// TIA Portal project "DATN" (V17)

(* hardware
DEVICE "S7-1200 station_1"  S7-1200 Station
   slot 0: "Rack_0"  S7-1200 Rack  Rack  V1.0
   slot 1: "PLC_1"  CPU 1214C DC/DC/DC  6ES7 214-1AG40-0XB0  V4.5
DEVICE "HMI_1"  KTP700 Basic PN
   slot 0: "HMI_1"  KTP700 Basic PN  6AV2 123-2GB03-0AX0  17.0.0.0
   slot 1: "HMI_RT_1"  KTP700 Basic PN  6AV2 123-2GB03-0AX0  17.0.0.0
   slot 5: "HMI_1.IE_CP_1"  PROFINET Interface  17.0.0.0
      slot 1: "PROFINET Interface_1"  PROFINET Interface
         slot 1: "Port_1"  Port
*)

// ===== PLC "PLC_1"  CPU 1214C DC/DC/DC =====

VAR_GLOBAL   // PLC tag table "Default tag table"
   "Tag_1" AT %M53.0 : Bool;
   "Reset_ctu_alarm" AT %M53.3 : Bool;
   "Tag_2" AT %M53.1 : Bool;
   "Tag_3" AT %M53.2 : Bool;
   "Error_lamp_alarm" AT %M53.4 : Bool;
   "time_up_maintenance" AT %M53.5 : Bool;
   "Alarm_not_product" AT %M53.6 : Bool;
   "Tag_4" AT %M100.0 : Bool;
   "Tag_5" AT %M100.1 : Bool;
   "Tag_6" AT %Q0.0 : Bool;
   "over_memory" AT %M54.0 : Bool;
   "stop_Sys_alarm" AT %M54.1 : Bool;
END_VAR

VAR_GLOBAL   // PLC tag table "Sensor"
   "Sensor_1" AT %I0.3 : Bool;
   "Sensor_2" AT %I0.4 : Bool;
   "Sensor_3" AT %I0.5 : Bool;
   "Sensor_4" AT %I0.6 : Bool;
   "Sensor_5" AT %I0.7 : Bool;
   "Sensor_Detech" AT %I0.2 : Bool;
END_VAR

VAR_GLOBAL   // PLC tag table "Output"
   "cylinder_1" AT %Q0.1 : Bool;
   "cylinder_2" AT %Q1.1 : Bool;
   "cylinder_3" AT %Q0.3 : Bool;
   "cylinder_4" AT %Q0.4 : Bool;
   "cylinder_5" AT %Q0.5 : Bool;
   "converyor" AT %Q1.0 : Bool;
   "led_error" AT %Q0.6 : Bool;
END_VAR

VAR_GLOBAL   // PLC tag table "Input_control"
   "Start" AT %I0.0 : Bool;
   "Stop" AT %I0.1 : Bool;
END_VAR

VAR_GLOBAL   // PLC tag table "State_system"
   "State_all" AT %M10.0 : Bool;
   "State_auto" AT %M10.1 : Bool;
END_VAR

VAR_GLOBAL   // PLC tag table "HMI"
   "hmi_manu_cylinder_1" AT %M10.3 : Bool;
   "hmi_manu_cylinder_2" AT %M10.4 : Bool;
   "hmi_manu_cylinder_3" AT %M10.5 : Bool;
   "hmi_manu_cylinder_4" AT %M10.6 : Bool;
   "hmi_manu_cylinder_5" AT %M10.7 : Bool;
   "hmi_active_count" AT %M11.0 : Bool;
   "HMI_ALARM" AT %M11.1 : Bool;
   "hmi_manu_conveyor" AT %M10.2 : Bool;
   "HMI_START" AT %M11.2 : Bool;
   "HMI_STOP" AT %M11.3 : Bool;
   "hmi_reset_count" AT %M11.4 : Bool;
   "hmi_problem_handled" AT %M11.5 : Bool;
   "hmi_reset_data" AT %M11.6 : Bool;
END_VAR

VAR_GLOBAL   // PLC tag table "Alarm"
   "Alarm1" AT %MW20 : Word;
   "Alarm1_Bit8_Motor_Fault" AT %M20.0 : Bool;   // Alarm motor Fault
   "Alarm1_Bit9_cylinder1_Fault" AT %M20.1 : Bool;   // Alarm cylinder1 Fault
   "Alarm1_Bit10_cylinder2_Fault" AT %M20.2 : Bool;   // Alarm cylinder2 Fault
   "Alarm1_Bit11_cylinder3_Fault" AT %M20.3 : Bool;   // Alarm cylinder3 Fault
   "Alarm1_Bit12_cylinder4_Fault" AT %M20.4 : Bool;   // Alarm cylinder4 Fault
   "Alarm1_Bit13_cylinder5_Fault" AT %M20.5 : Bool;   // Alarm cylinder5 Fault
   "Alarm1_Bit14" AT %M20.6 : Bool;   // Spare
   "Alarm1_Bit15" AT %M20.7 : Bool;   // Spare
   "Alarm1_Bit0" AT %M21.0 : Bool;   // Spare
   "Alarm1_Bit1" AT %M21.1 : Bool;   // Spare
   "Alarm1_Bit2" AT %M21.2 : Bool;   // Spare
   "Alarm1_Bit3" AT %M21.3 : Bool;   // Spare
   "Alarm_over_memory" AT %M21.4 : Bool;   // over memory
   "Alarm_emergence_stop_web" AT %M21.5 : Bool;   // emergence stop
   "Alarm_camera_error" AT %M21.6 : Bool;   // camera error
   "Alarm_maintenance_time" AT %M21.7 : Bool;   // up to maintenance time
END_VAR

VAR_GLOBAL   // PLC tag table "Simulater"
   "Sim_motor_tripped" AT %M52.0 : Bool;
   "Sim_cylinder1_tripped" AT %M52.1 : Bool;
   "Sim_cylinder2_tripped" AT %M52.2 : Bool;
   "Sim_cylinder3_tripped" AT %M52.3 : Bool;
   "Sim_cylinder4_tripped" AT %M52.4 : Bool;
   "Sim_cylinder5_tripped" AT %M52.5 : Bool;
END_VAR

DATA_BLOCK "Array_threading"   // DB1
{ S7_Optimized_Access := 'FALSE' }
VERSION : 0.1
   VAR
      array_threading_1 : Array[0..20] of Int;
      array_threading_2 : Array[0..20] of Int;
      array_threading_3 : Array[0..20] of Int;
      array_threading_4 : Array[0..20] of Int;
      array_threading_5 : Array[0..20] of Int;
      last_run_1 : Bool;
      last_run_2 : Bool;
      last_run_3 : Bool;
      last_run_4 : Bool;
      last_run_5 : Bool;
   END_VAR
BEGIN
END_DATA_BLOCK

DATA_BLOCK "Data_webcam"   // DB7
{ S7_Optimized_Access := 'FALSE' }
VERSION : 0.1
   VAR
      new_position : Int;
      save_new_position : Bool;
      state_camera : Bool := true;
      alarm_error : Bool;
      state_auto : Bool;
      last_state_sensor_1 : Bool;
      last_state_sensor_2 : Bool;
      last_state_sensor_3 : Bool;
      last_state_sensor_4 : Bool;
      last_state_sensor_5 : Bool;
      last_save_new_position : Bool;
   END_VAR
BEGIN
END_DATA_BLOCK

DATA_BLOCK "Data_count_Position"   // DB8
{ S7_Optimized_Access := 'FALSE' }
VERSION : 0.1
   VAR
      Adress_1 : Real;
      Adress_2 : Real;
      Adress_3 : Real;
      Adress_4 : Real;
      Adress_5 : Real;
      Adress_6 : Real;
   END_VAR
BEGIN
END_DATA_BLOCK

DATA_BLOCK "Data_alarm"   // DB17
{ S7_Optimized_Access := 'FALSE' }
VERSION : 0.1
   VAR
      Motor_tripped : Bool;
      Cylinder1_tripped : Bool;
      Cylinder2_tripped : Bool;
      Cylinder3_tripped : Bool;
      Cylinder4_tripped : Bool;
      Cylinder5_tripped : Bool;
      Camera_tripped : Bool;
      Time_to_Maintenance : DInt;
   END_VAR
BEGIN
END_DATA_BLOCK

DATA_BLOCK "state_to_webserver"   // DB22
{ S7_Optimized_Access := 'FALSE' }
VERSION : 0.1
   VAR
      state_sensor_1 : Bool;
      state_sensor_2 : Bool;
      state_sensor_3 : Bool;
      state_sensor_4 : Bool;
      state_sensor_5 : Bool;
      state_sensor_detech : Bool;
      state_emergency_stop : Bool;
      state_cylinder_1 : Int;
      state_cylinder_2 : Int;
      state_cylinder_3 : Int;
      state_cylinder_4 : Int;
      state_cylinder_5 : Int;
      state_motor : Int;
      state_auto : Int;
   END_VAR
BEGIN
END_DATA_BLOCK

// folder: System blocks/Program resources

DATA_BLOCK "IEC_Timer_0_DB"   // DB2
{ S7_Optimized_Access := 'TRUE' }
AUTHOR : Simatic
FAMILY : IEC
NAME : IEC_TMR
VERSION : 1.0
// stored: InstanceOfName IEC_TIMER
"IEC_TIMER"
BEGIN
END_DATA_BLOCK

DATA_BLOCK "IEC_Timer_0_DB_1"   // DB3
{ S7_Optimized_Access := 'TRUE' }
AUTHOR : Simatic
FAMILY : IEC
NAME : IEC_TMR
VERSION : 1.0
// stored: InstanceOfName IEC_TIMER
"IEC_TIMER"
BEGIN
END_DATA_BLOCK

DATA_BLOCK "IEC_Timer_0_DB_2"   // DB4
{ S7_Optimized_Access := 'TRUE' }
AUTHOR : Simatic
FAMILY : IEC
NAME : IEC_TMR
VERSION : 1.0
// stored: InstanceOfName IEC_TIMER
"IEC_TIMER"
BEGIN
END_DATA_BLOCK

DATA_BLOCK "IEC_Timer_0_DB_3"   // DB5
{ S7_Optimized_Access := 'TRUE' }
AUTHOR : Simatic
FAMILY : IEC
NAME : IEC_TMR
VERSION : 1.0
// stored: InstanceOfName IEC_TIMER
"IEC_TIMER"
BEGIN
END_DATA_BLOCK

DATA_BLOCK "IEC_Timer_0_DB_4"   // DB6
{ S7_Optimized_Access := 'TRUE' }
AUTHOR : Simatic
FAMILY : IEC
NAME : IEC_TMR
VERSION : 1.0
// stored: InstanceOfName IEC_TIMER
"IEC_TIMER"
BEGIN
END_DATA_BLOCK

DATA_BLOCK "IEC_Counter_0_DB"   // DB9
{ S7_Optimized_Access := 'FALSE' }
AUTHOR : Simatic
FAMILY : IEC
NAME : CNTR
VERSION : 1.0
// stored: InstanceOfName IEC_COUNTER
"IEC_COUNTER"
BEGIN
END_DATA_BLOCK

DATA_BLOCK "IEC_Counter_0_DB_1"   // DB10
{ S7_Optimized_Access := 'TRUE' }
AUTHOR : Simatic
FAMILY : IEC
NAME : CNTR
VERSION : 1.0
// stored: InstanceOfName IEC_COUNTER
"IEC_COUNTER"
BEGIN
END_DATA_BLOCK

DATA_BLOCK "IEC_Counter_0_DB_2"   // DB11
{ S7_Optimized_Access := 'TRUE' }
AUTHOR : Simatic
FAMILY : IEC
NAME : CNTR
VERSION : 1.0
// stored: InstanceOfName IEC_COUNTER
"IEC_COUNTER"
BEGIN
END_DATA_BLOCK

DATA_BLOCK "IEC_Counter_0_DB_3"   // DB12
{ S7_Optimized_Access := 'TRUE' }
AUTHOR : Simatic
FAMILY : IEC
NAME : CNTR
VERSION : 1.0
// stored: InstanceOfName IEC_COUNTER
"IEC_COUNTER"
BEGIN
END_DATA_BLOCK

DATA_BLOCK "IEC_Counter_0_DB_4"   // DB13
{ S7_Optimized_Access := 'TRUE' }
AUTHOR : Simatic
FAMILY : IEC
NAME : CNTR
VERSION : 1.0
// stored: InstanceOfName IEC_COUNTER
"IEC_COUNTER"
BEGIN
END_DATA_BLOCK

DATA_BLOCK "IEC_Timer_0_DB_7"   // DB14
{ S7_Optimized_Access := 'TRUE' }
AUTHOR : Simatic
FAMILY : IEC
NAME : IEC_TMR
VERSION : 1.0
// stored: InstanceOfName IEC_TIMER
"IEC_TIMER"
BEGIN
END_DATA_BLOCK

DATA_BLOCK "IEC_Counter_0_DB_6"   // DB20
{ S7_Optimized_Access := 'TRUE' }
AUTHOR : SIMATIC
FAMILY : IEC
NAME : DCNTR
VERSION : 1.2
// stored: InstanceOfName IEC_DCOUNTER
"IEC_DCOUNTER"
BEGIN
END_DATA_BLOCK

DATA_BLOCK "IEC_Timer_0_DB_9"   // DB21
{ S7_Optimized_Access := 'TRUE' }
AUTHOR : Simatic
FAMILY : IEC
NAME : IEC_TMR
VERSION : 1.0
// stored: InstanceOfName IEC_TIMER
"IEC_TIMER"
BEGIN
END_DATA_BLOCK

// folder: (top level)

FUNCTION "Auto" : Void   // FC1, LAD
{ S7_Optimized_Access := 'TRUE' }
VERSION : 0.1
   VAR_INPUT
      error_alarm : Bool;
      new_position : Int;
      save_new_position : Bool;
      reset_data : Bool;
      sensor_1 : Bool;
      sensor_2 : Bool;
      sensor_3 : Bool;
      sensor_4 : Bool;
      sensor_5 : Bool;
   END_VAR
   VAR_OUTPUT
      cylinder_1 : Bool;
      cylinder_2 : Bool;
      cylinder_3 : Bool;
      cylinder_4 : Bool;
      cylinder_5 : Bool;
      over_memory : Bool;
   END_VAR
   VAR_TEMP
      loop_element : Int;
      last_child_array_1 : Int;
      last_child_array_2 : Int;
      last_child_array_3 : Int;
      last_child_array_4 : Int;
      last_child_array_5 : Int;
      trigger_sensor_1 : Bool;
      trigger_sensor_2 : Bool;
      trigger_sensor_3 : Bool;
      trigger_sensor_4 : Bool;
      trigger_sensor_5 : Bool;
   END_VAR
BEGIN

REGION Network 1 (SCL): Program main
   // chuong trinh dieu khien
   // ========================
   // Reset trạng thái khi save_new_position = 0 hoặc cảm biến = 0
   // ========================
   IF #save_new_position = FALSE THEN
       "Data_webcam".last_save_new_position := FALSE;
   END_IF;

   IF #sensor_1 = FALSE THEN
       "Data_webcam".last_state_sensor_1 := FALSE;
   END_IF;

   IF #sensor_2 = FALSE THEN
       "Data_webcam".last_state_sensor_2 := FALSE;
   END_IF;

   IF #sensor_3 = FALSE THEN
       "Data_webcam".last_state_sensor_3 := FALSE;
   END_IF;

   IF #sensor_4 = FALSE THEN
       "Data_webcam".last_state_sensor_4 := FALSE;
   END_IF;

   IF #sensor_5 = FALSE THEN
       "Data_webcam".last_state_sensor_5 := FALSE;
   END_IF;

   // ========================
   // Xử lý khi có sản phẩm mới
   // ========================
   IF (#save_new_position = TRUE) AND ("Data_webcam".last_save_new_position = FALSE) AND (#error_alarm = False) THEN
       "Data_webcam".last_save_new_position := TRUE;

       // Tìm vị trí cuối cùng của mỗi mảng
       #last_child_array_1 := -1;
       #last_child_array_2 := -1;
       #last_child_array_3 := -1;
       #last_child_array_4 := -1;
       #last_child_array_5 := -1;

       FOR #loop_element := 0 TO 20 DO
           IF ("Array_threading".array_threading_1[#loop_element] = 1) OR ("Array_threading".array_threading_1[#loop_element] = 2) THEN
               #last_child_array_1 := #loop_element;
           END_IF;
           IF ("Array_threading".array_threading_2[#loop_element] = 1) OR ("Array_threading".array_threading_2[#loop_element] = 2) THEN
               #last_child_array_2 := #loop_element;
           END_IF;
           IF ("Array_threading".array_threading_3[#loop_element] = 1) OR ("Array_threading".array_threading_3[#loop_element] = 2) THEN
               #last_child_array_3 := #loop_element;
           END_IF;
           IF ("Array_threading".array_threading_4[#loop_element] = 1) OR ("Array_threading".array_threading_4[#loop_element] = 2) THEN
               #last_child_array_4 := #loop_element;
           END_IF;
           IF ("Array_threading".array_threading_5[#loop_element] = 1) OR ("Array_threading".array_threading_5[#loop_element] = 2) THEN
               #last_child_array_5 := #loop_element;
           END_IF;
       END_FOR;

       // Gán vị trí mới (tránh tràn mảng)
       CASE #new_position OF
           1:
               IF #last_child_array_1 < 20 THEN
                   "Array_threading".array_threading_1[#last_child_array_1 + 1] := 1;
               END_IF;

           2:
               IF #last_child_array_1 < 20 AND #last_child_array_2 < 20 THEN
                   "Array_threading".array_threading_1[#last_child_array_1 + 1] := 2;
                   "Array_threading".array_threading_2[#last_child_array_2 + 1] := 1;
               END_IF;

           3:
               IF #last_child_array_1 < 20 AND #last_child_array_2 < 20 AND #last_child_array_3 < 20 THEN
                   "Array_threading".array_threading_1[#last_child_array_1 + 1] := 2;
                   "Array_threading".array_threading_2[#last_child_array_2 + 1] := 2;
                   "Array_threading".array_threading_3[#last_child_array_3 + 1] := 1;
               END_IF;

           4:
               IF #last_child_array_1 < 20 AND #last_child_array_2 < 20 AND
                   #last_child_array_3 < 20 AND #last_child_array_4 < 20 THEN
                   "Array_threading".array_threading_1[#last_child_array_1 + 1] := 2;
                   "Array_threading".array_threading_2[#last_child_array_2 + 1] := 2;
                   "Array_threading".array_threading_3[#last_child_array_3 + 1] := 2;
                   "Array_threading".array_threading_4[#last_child_array_4 + 1] := 1;
               END_IF;

           5:
               IF #last_child_array_1 < 20 AND #last_child_array_2 < 20 AND
                   #last_child_array_3 < 20 AND #last_child_array_4 < 20 AND
                   #last_child_array_5 < 20 THEN
                   "Array_threading".array_threading_1[#last_child_array_1 + 1] := 2;
                   "Array_threading".array_threading_2[#last_child_array_2 + 1] := 2;
                   "Array_threading".array_threading_3[#last_child_array_3 + 1] := 2;
                   "Array_threading".array_threading_4[#last_child_array_4 + 1] := 2;
                   "Array_threading".array_threading_5[#last_child_array_5 + 1] := 1;
               END_IF;

           6:
               IF #last_child_array_1 < 20 AND #last_child_array_2 < 20 AND
                   #last_child_array_3 < 20 AND #last_child_array_4 < 20 AND
                   #last_child_array_5 < 20 THEN
                   "Array_threading".array_threading_1[#last_child_array_1 + 1] := 2;
                   "Array_threading".array_threading_2[#last_child_array_2 + 1] := 2;
                   "Array_threading".array_threading_3[#last_child_array_3 + 1] := 2;
                   "Array_threading".array_threading_4[#last_child_array_4 + 1] := 2;
                   "Array_threading".array_threading_5[#last_child_array_5 + 1] := 2;
               END_IF;
       END_CASE;
   END_IF;

   // Báo tràn bộ nhớ phân loại
   IF #last_child_array_1 = 20 OR #last_child_array_2 = 20 OR
       #last_child_array_3 = 20 OR #last_child_array_4 = 20 OR
       #last_child_array_5 = 20 THEN
       #over_memory := TRUE;
   END_IF;

   // ========================
   // Xử lý từng cảm biến khi phát hiện sản phẩm
   // ========================
   // ==== SENSOR 1 ====
   IF (#sensor_1 = TRUE) AND (#sensor_1 <> "Data_webcam".last_state_sensor_1) AND "Array_threading".last_run_1 = FALSE THEN
       // Set trigger cho TOF

       IF "Array_threading".array_threading_1[0] = 1 THEN
           #trigger_sensor_1 := TRUE;
       END_IF;

       FOR #loop_element := 0 TO 19 DO
           "Array_threading".array_threading_1[#loop_element] := "Array_threading".array_threading_1[#loop_element + 1];
       END_FOR;
       "Array_threading".array_threading_1[20] := 0;
       "Data_webcam".last_state_sensor_1 := TRUE;
   END_IF;

   // ==== SENSOR 2 ====
   IF (#sensor_2 = TRUE) AND (#sensor_2 <> "Data_webcam".last_state_sensor_2) AND "Array_threading".last_run_2 = FALSE THEN
       IF "Array_threading".array_threading_2[0] = 1 THEN
           #trigger_sensor_2 := TRUE;
       END_IF;

       FOR #loop_element := 0 TO 19 DO
           "Array_threading".array_threading_2[#loop_element] := "Array_threading".array_threading_2[#loop_element + 1];
       END_FOR;
       "Array_threading".array_threading_2[20] := 0;
       "Data_webcam".last_state_sensor_2 := TRUE;
   END_IF;

   // ==== SENSOR 3 ====
   IF (#sensor_3 = TRUE) AND (#sensor_3 <> "Data_webcam".last_state_sensor_3) AND "Array_threading".last_run_3 = FALSE THEN
       IF "Array_threading".array_threading_3[0] = 1 THEN
           #trigger_sensor_3 := TRUE;
       END_IF;

       FOR #loop_element := 0 TO 19 DO
           "Array_threading".array_threading_3[#loop_element] := "Array_threading".array_threading_3[#loop_element + 1];
       END_FOR;
       "Array_threading".array_threading_3[20] := 0;
       "Data_webcam".last_state_sensor_3 := TRUE;
   END_IF;

   // ==== SENSOR 4 ====
   IF (#sensor_4 = TRUE) AND (#sensor_4 <> "Data_webcam".last_state_sensor_4) AND "Array_threading".last_run_4 = FALSE THEN
       IF "Array_threading".array_threading_4[0] = 1 THEN
           #trigger_sensor_4 := TRUE;
       END_IF;

       FOR #loop_element := 0 TO 19 DO
           "Array_threading".array_threading_4[#loop_element] := "Array_threading".array_threading_4[#loop_element + 1];
       END_FOR;
       "Array_threading".array_threading_4[20] := 0;
       "Data_webcam".last_state_sensor_4 := TRUE;
   END_IF;

   // ==== SENSOR 5 ====
   IF (#sensor_5 = TRUE) AND (#sensor_5 <> "Data_webcam".last_state_sensor_5) AND "Array_threading".last_run_5 = FALSE THEN
       IF "Array_threading".array_threading_5[0] = 1 THEN
           #trigger_sensor_5 := TRUE;
       END_IF;

       FOR #loop_element := 0 TO 19 DO
           "Array_threading".array_threading_5[#loop_element] := "Array_threading".array_threading_5[#loop_element + 1];
       END_FOR;
       "Array_threading".array_threading_5[20] := 0;
       "Data_webcam".last_state_sensor_5 := TRUE;
   END_IF;

   // ======== TIMER ON DELAY ========
   "IEC_Timer_0_DB".TOF(IN:=#trigger_sensor_1,PT:=T#3s);
   "IEC_Timer_0_DB_1".TOF(IN:=#trigger_sensor_2,PT:=T#3s);
   "IEC_Timer_0_DB_2".TOF(IN :=#trigger_sensor_3,PT := T#3s);
   "IEC_Timer_0_DB_3".TOF(IN :=#trigger_sensor_4,PT:=T#3s);
   "IEC_Timer_0_DB_4".TOF(IN:=#trigger_sensor_5,PT:=T#3s);

   IF ("IEC_Timer_0_DB".ET >= T#1s) AND ("IEC_Timer_0_DB".ET < T#2s) THEN
       #cylinder_1 := TRUE;
   ELSE
       #cylinder_1 := FALSE;
   END_IF;

   IF ("IEC_Timer_0_DB_1".ET >= T#1s) AND ("IEC_Timer_0_DB_1".ET < T#2s) THEN
       #cylinder_2 := TRUE;
   ELSE
       #cylinder_2 := FALSE;
   END_IF;

   IF ("IEC_Timer_0_DB_2".ET >= T#1s) AND ("IEC_Timer_0_DB_2".ET < T#2s) THEN
       #cylinder_3 := TRUE;
   ELSE
       #cylinder_3 := FALSE;
   END_IF;

   IF ("IEC_Timer_0_DB_3".ET >= T#1s) AND ("IEC_Timer_0_DB_3".ET < T#2s) THEN
       #cylinder_4 := TRUE;
   ELSE
       #cylinder_4 := FALSE;
   END_IF;

   IF ("IEC_Timer_0_DB_4".ET >= T#1s) AND ("IEC_Timer_0_DB_4".ET < T#2s) THEN
       #cylinder_5 := TRUE;
   ELSE
       #cylinder_5 := FALSE;
   END_IF;


   // ======== RESET DATA  ========
   IF #reset_data = TRUE THEN
       FOR #loop_element := 0 TO 20 DO
           "Array_threading".array_threading_1[#loop_element] := 0;
           "Array_threading".array_threading_2[#loop_element] := 0;
           "Array_threading".array_threading_3[#loop_element] := 0;
           "Array_threading".array_threading_4[#loop_element] := 0;
           "Array_threading".array_threading_5[#loop_element] := 0;
       END_FOR;
   END_IF;
END_REGION
END_FUNCTION

FUNCTION "Manual" : Void   // FC2, LAD
{ S7_Optimized_Access := 'TRUE' }
VERSION : 0.1
   VAR_INPUT
      control_conveyor : Bool;
      control_cylinder_1 : Bool;
      control_cylinder_2 : Bool;
      control_cylinder_3 : Bool;
      control_cylinder_4 : Bool;
      control_cylinder_5 : Bool;
   END_VAR
   VAR_OUTPUT
      conveyor : Bool;
      cylinder_1 : Bool;
      cylinder_2 : Bool;
      cylinder_3 : Bool;
      cylinder_4 : Bool;
      cylinder_5 : Bool;
   END_VAR
BEGIN

REGION Network 1: Program manual conveyor
   // chuong trinh dieu khien bang tay bang tai
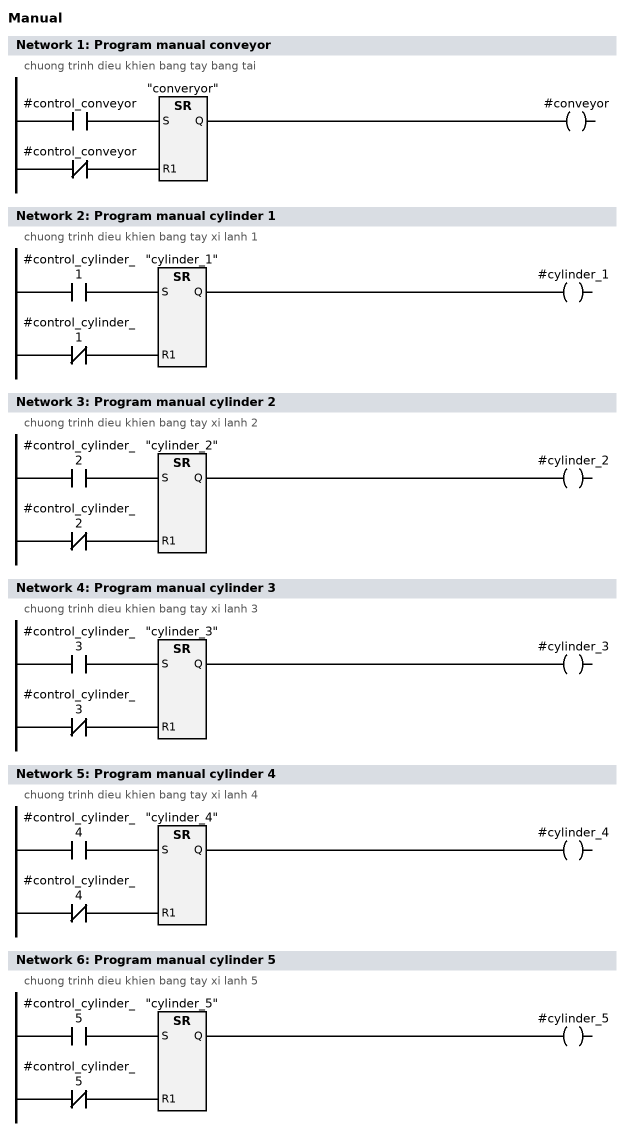
   RUNG wire#powerrail
      Contact( #control_conveyor )
      S_SR(operand := "converyor", r1 := wire#w1)
      Coil( #conveyor )
   END_RUNG
   RUNG wire#powerrail
      I_Contact( #control_conveyor )
   END_RUNG wire#w1
   // the same network as SCL:
   IF #control_conveyor THEN
       "converyor" := TRUE;   // SR flip-flop
   END_IF;
   IF NOT #control_conveyor THEN "converyor" := FALSE; END_IF;
   #conveyor := "converyor";
END_REGION

REGION Network 2: Program manual cylinder 1
   // chuong trinh dieu khien bang tay xi lanh 1
   RUNG wire#powerrail
      Contact( #control_cylinder_1 )
      S_SR(operand := "cylinder_1", r1 := wire#w1)
      Coil( #cylinder_1 )
   END_RUNG
   RUNG wire#powerrail
      I_Contact( #control_cylinder_1 )
   END_RUNG wire#w1
   // the same network as SCL:
   IF #control_cylinder_1 THEN
       "cylinder_1" := TRUE;   // SR flip-flop
   END_IF;
   IF NOT #control_cylinder_1 THEN "cylinder_1" := FALSE; END_IF;
   #cylinder_1 := "cylinder_1";
END_REGION

REGION Network 3: Program manual cylinder 2
   // chuong trinh dieu khien bang tay xi lanh 2
   RUNG wire#powerrail
      Contact( #control_cylinder_2 )
      S_SR(operand := "cylinder_2", r1 := wire#w1)
      Coil( #cylinder_2 )
   END_RUNG
   RUNG wire#powerrail
      I_Contact( #control_cylinder_2 )
   END_RUNG wire#w1
   // the same network as SCL:
   IF #control_cylinder_2 THEN
       "cylinder_2" := TRUE;   // SR flip-flop
   END_IF;
   IF NOT #control_cylinder_2 THEN "cylinder_2" := FALSE; END_IF;
   #cylinder_2 := "cylinder_2";
END_REGION

REGION Network 4: Program manual cylinder 3
   // chuong trinh dieu khien bang tay xi lanh 3
   RUNG wire#powerrail
      Contact( #control_cylinder_3 )
      S_SR(operand := "cylinder_3", r1 := wire#w1)
      Coil( #cylinder_3 )
   END_RUNG
   RUNG wire#powerrail
      I_Contact( #control_cylinder_3 )
   END_RUNG wire#w1
   // the same network as SCL:
   IF #control_cylinder_3 THEN
       "cylinder_3" := TRUE;   // SR flip-flop
   END_IF;
   IF NOT #control_cylinder_3 THEN "cylinder_3" := FALSE; END_IF;
   #cylinder_3 := "cylinder_3";
END_REGION

REGION Network 5: Program manual cylinder 4
   // chuong trinh dieu khien bang tay xi lanh 4
   RUNG wire#powerrail
      Contact( #control_cylinder_4 )
      S_SR(operand := "cylinder_4", r1 := wire#w1)
      Coil( #cylinder_4 )
   END_RUNG
   RUNG wire#powerrail
      I_Contact( #control_cylinder_4 )
   END_RUNG wire#w1
   // the same network as SCL:
   IF #control_cylinder_4 THEN
       "cylinder_4" := TRUE;   // SR flip-flop
   END_IF;
   IF NOT #control_cylinder_4 THEN "cylinder_4" := FALSE; END_IF;
   #cylinder_4 := "cylinder_4";
END_REGION

REGION Network 6: Program manual cylinder 5
   // chuong trinh dieu khien bang tay xi lanh 5
   RUNG wire#powerrail
      Contact( #control_cylinder_5 )
      S_SR(operand := "cylinder_5", r1 := wire#w1)
      Coil( #cylinder_5 )
   END_RUNG
   RUNG wire#powerrail
      I_Contact( #control_cylinder_5 )
   END_RUNG wire#w1
   // the same network as SCL:
   IF #control_cylinder_5 THEN
       "cylinder_5" := TRUE;   // SR flip-flop
   END_IF;
   IF NOT #control_cylinder_5 THEN "cylinder_5" := FALSE; END_IF;
   #cylinder_5 := "cylinder_5";
END_REGION
END_FUNCTION

FUNCTION "Count_Position" : Void   // FC3, LAD
{ S7_Optimized_Access := 'TRUE' }
VERSION : 0.1
   VAR_INPUT
      Postion_1 : Bool;
      Position_2 : Bool;
      Position_3 : Bool;
      Position_4 : Bool;
      Position_5 : Bool;
      Reset_count : Bool;
      Actice_count : Bool;
   END_VAR
BEGIN

REGION Network 1: Count position 1
   // Đếm vị trí phân loại 1
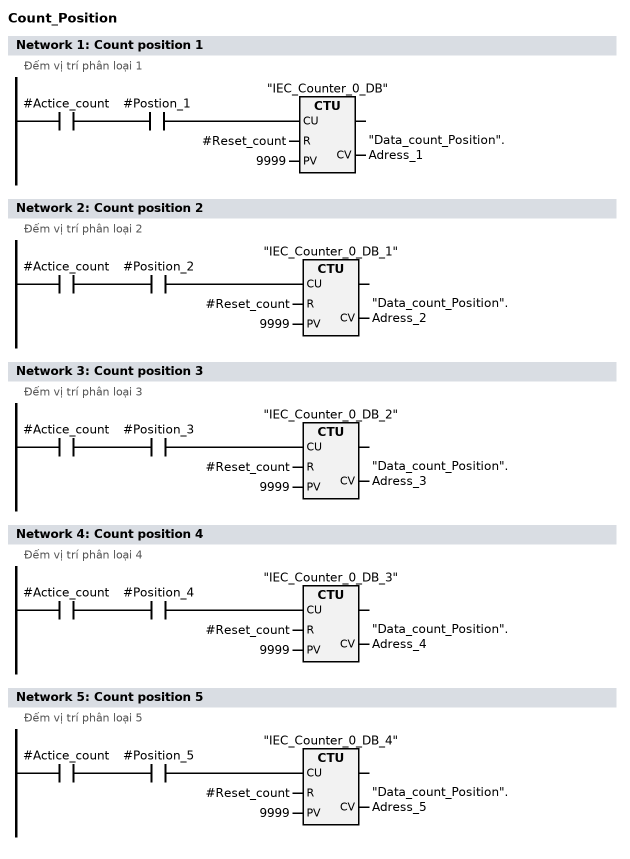
   "IEC_Counter_0_DB".CTU(CU := #Actice_count AND #Postion_1,
                          R := #Reset_count,
                          PV := 9999,
                          CV => "Data_count_Position".Adress_1);
END_REGION

REGION Network 2: Count position 2
   // Đếm vị trí phân loại 2
   "IEC_Counter_0_DB_1".CTU(CU := #Actice_count AND #Position_2,
                           R := #Reset_count,
                           PV := 9999,
                           CV => "Data_count_Position".Adress_2);
END_REGION

REGION Network 3: Count position 3
   // Đếm vị trí phân loại 3
   "IEC_Counter_0_DB_2".CTU(CU := #Actice_count AND #Position_3,
                           R := #Reset_count,
                           PV := 9999,
                           CV => "Data_count_Position".Adress_3);
END_REGION

REGION Network 4: Count position 4
   // Đếm vị trí phân loại 4
   "IEC_Counter_0_DB_3".CTU(CU := #Actice_count AND #Position_4,
                           R := #Reset_count,
                           PV := 9999,
                           CV => "Data_count_Position".Adress_4);
END_REGION

REGION Network 5: Count position 5
   // Đếm vị trí phân loại 5
   "IEC_Counter_0_DB_4".CTU(CU := #Actice_count AND #Position_5,
                           R := #Reset_count,
                           PV := 9999,
                           CV => "Data_count_Position".Adress_5);
END_REGION
END_FUNCTION

FUNCTION "Alarm" : Void   // FC4, LAD
{ S7_Optimized_Access := 'TRUE' }
VERSION : 0.1
   VAR_INPUT
      I_Alarm_simulater : Bool;
   END_VAR
   VAR_OUTPUT
      Alarm1_Bit8_Motor_Fault : Bool;
      Alarm1_Bit9_cylinder1_Fault : Bool;
      Alarm1_Bit10_cylinder2_Fault : Bool;
      Alarm1_Bit11_cylinder3_Fault : Bool;
      Alarm1_Bit12_cylinder4_Fault : Bool;
      Alarm1_Bit13_cylinder5_Fault : Bool;
      state_error : Bool;
      Stop_sys : Bool;
   END_VAR
   VAR_TEMP
      count : Int;
      loop_element : Int;
   END_VAR
BEGIN

REGION Network 1: Alarm program
   // chuong trinh alarm
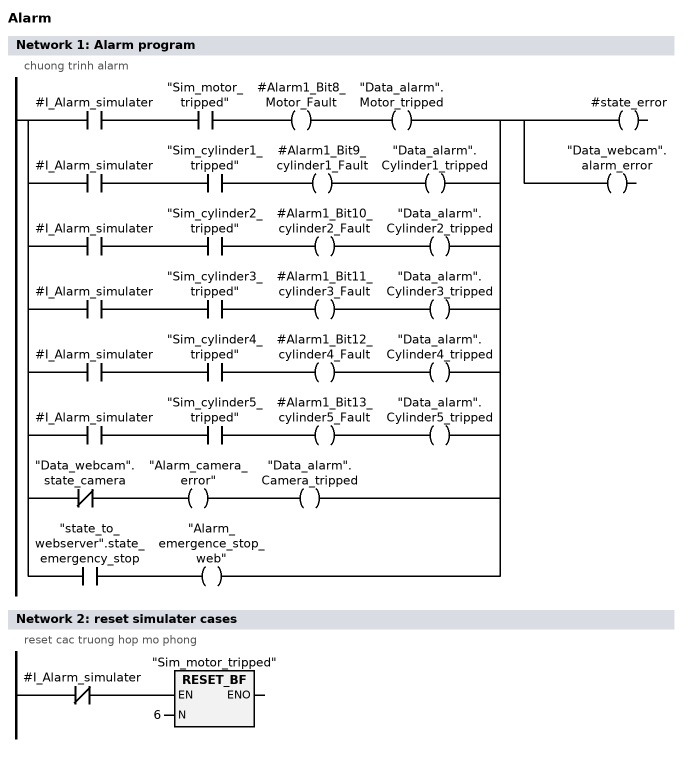
   RUNG wire#powerrail
      Contact( #I_Alarm_simulater )
      Contact( "Sim_motor_tripped" )
      Coil( #Alarm1_Bit8_Motor_Fault )
      Coil( "Data_alarm".Motor_tripped )
      wire#w1
      Coil( #state_error )
   END_RUNG
   RUNG wire#powerrail
      Contact( #I_Alarm_simulater )
      Contact( "Sim_cylinder1_tripped" )
      Coil( #Alarm1_Bit9_cylinder1_Fault )
      Coil( "Data_alarm".Cylinder1_tripped )
   END_RUNG wire#w1
   RUNG wire#powerrail
      Contact( #I_Alarm_simulater )
      Contact( "Sim_cylinder2_tripped" )
      Coil( #Alarm1_Bit10_cylinder2_Fault )
      Coil( "Data_alarm".Cylinder2_tripped )
   END_RUNG wire#w1
   RUNG wire#powerrail
      Contact( #I_Alarm_simulater )
      Contact( "Sim_cylinder3_tripped" )
      Coil( #Alarm1_Bit11_cylinder3_Fault )
      Coil( "Data_alarm".Cylinder3_tripped )
   END_RUNG wire#w1
   RUNG wire#powerrail
      Contact( #I_Alarm_simulater )
      Contact( "Sim_cylinder4_tripped" )
      Coil( #Alarm1_Bit12_cylinder4_Fault )
      Coil( "Data_alarm".Cylinder4_tripped )
   END_RUNG wire#w1
   RUNG wire#powerrail
      Contact( #I_Alarm_simulater )
      Contact( "Sim_cylinder5_tripped" )
      Coil( #Alarm1_Bit13_cylinder5_Fault )
      Coil( "Data_alarm".Cylinder5_tripped )
   END_RUNG wire#w1
   RUNG wire#powerrail
      I_Contact( "Data_webcam".state_camera )
      Coil( "Alarm_camera_error" )
      Coil( "Data_alarm".Camera_tripped )
   END_RUNG wire#w1
   RUNG wire#powerrail
      Contact( "state_to_webserver".state_emergency_stop )
      Coil( "Alarm_emergence_stop_web" )
   END_RUNG wire#w1
   RUNG wire#w1
      Coil( "Data_webcam".alarm_error )
   END_RUNG
   // the same network as SCL:
   #Alarm1_Bit8_Motor_Fault := #I_Alarm_simulater AND "Sim_motor_tripped";
   "Data_alarm".Motor_tripped := #Alarm1_Bit8_Motor_Fault;
   #Alarm1_Bit9_cylinder1_Fault := #I_Alarm_simulater AND "Sim_cylinder1_tripped";
   "Data_alarm".Cylinder1_tripped := #Alarm1_Bit9_cylinder1_Fault;
   #Alarm1_Bit10_cylinder2_Fault := #I_Alarm_simulater AND "Sim_cylinder2_tripped";
   "Data_alarm".Cylinder2_tripped := #Alarm1_Bit10_cylinder2_Fault;
   #Alarm1_Bit11_cylinder3_Fault := #I_Alarm_simulater AND "Sim_cylinder3_tripped";
   "Data_alarm".Cylinder3_tripped := #Alarm1_Bit11_cylinder3_Fault;
   #Alarm1_Bit12_cylinder4_Fault := #I_Alarm_simulater AND "Sim_cylinder4_tripped";
   "Data_alarm".Cylinder4_tripped := #Alarm1_Bit12_cylinder4_Fault;
   #Alarm1_Bit13_cylinder5_Fault := #I_Alarm_simulater AND "Sim_cylinder5_tripped";
   "Data_alarm".Cylinder5_tripped := #Alarm1_Bit13_cylinder5_Fault;
   "Alarm_camera_error" := NOT "Data_webcam".state_camera;
   "Data_alarm".Camera_tripped := NOT "Data_webcam".state_camera;
   "Alarm_emergence_stop_web" := "state_to_webserver".state_emergency_stop;
   #state_error := #Alarm1_Bit8_Motor_Fault OR #Alarm1_Bit9_cylinder1_Fault OR #Alarm1_Bit10_cylinder2_Fault OR #Alarm1_Bit11_cylinder3_Fault OR #Alarm1_Bit12_cylinder4_Fault OR #Alarm1_Bit13_cylinder5_Fault OR NOT "Data_webcam".state_camera OR "state_to_webserver".state_emergency_stop;
   "Data_webcam".alarm_error := #state_error;
END_REGION

REGION Network 2: reset simulater cases
   // reset cac truong hop mo phong
   // no SCL statement known for RBitfield: written as a call
   IF NOT #I_Alarm_simulater THEN RESET_BF(operand := "Sim_motor_tripped", n := 6); END_IF;
END_REGION

REGION Network 3 (SCL): troubleshoot system
   // Xử lí sự cố
   IF  (#Alarm1_Bit9_cylinder1_Fault = FALSE) AND
       (#Alarm1_Bit10_cylinder2_Fault = FALSE) AND
       (#Alarm1_Bit11_cylinder3_Fault = FALSE) AND
       (#Alarm1_Bit12_cylinder4_Fault = FALSE) AND
       (#Alarm1_Bit13_cylinder5_Fault = FALSE) THEN
       "Array_threading".last_run_1 := FALSE;
       "Array_threading".last_run_2 := FALSE;
       "Array_threading".last_run_3 := FALSE;
       "Array_threading".last_run_4 := FALSE;
       "Array_threading".last_run_5 := FALSE;
   ELSE
       IF "Array_threading".array_threading_1[0] = 0 AND "Array_threading".array_threading_2[0] = 0 AND
           "Array_threading".array_threading_3[0] = 0 AND "Array_threading".array_threading_4[0] = 0 AND
           "Array_threading".array_threading_5[0] = 0 THEN
           #Stop_sys := True;
       END_IF;
   END_IF;

   // Kiểm tra motor lỗi
   IF #Alarm1_Bit8_Motor_Fault = TRUE THEN
       #Stop_sys := TRUE;
       // Kiểm tra xi lanh 1
   ELSIF #Alarm1_Bit9_cylinder1_Fault = TRUE THEN
       IF "Array_threading".array_threading_1[0] = 1 THEN
           "Array_threading".last_run_1 := True;
       END_IF;

       IF "Array_threading".last_run_1 = TRUE AND "Sensor_1" = TRUE THEN
           #Stop_sys := True;
       END_IF;
       // Kiểm tra xi lanh 2
   ELSIF #Alarm1_Bit10_cylinder2_Fault = TRUE THEN
       IF "Array_threading".array_threading_2[0] = 1 THEN
           "Array_threading".last_run_2 := True;
       END_IF;

       IF "Array_threading".last_run_2 = TRUE AND "Sensor_2" = TRUE THEN
           #Stop_sys := True;
       END_IF;
   // Kiểm tra xi lanh 3
   ELSIF #Alarm1_Bit11_cylinder3_Fault = TRUE THEN
       IF "Array_threading".array_threading_3[0] = 1 THEN
           "Array_threading".last_run_3 := True;
       END_IF;

       IF "Array_threading".last_run_3 = TRUE AND "Sensor_3" = TRUE THEN
           #Stop_sys := True;
       END_IF;
   // Kiểm tra xi lanh 4
   ELSIF #Alarm1_Bit12_cylinder4_Fault = TRUE THEN
       IF "Array_threading".array_threading_4[0] = 1 THEN
           "Array_threading".last_run_4 := True;
       END_IF;

       IF "Array_threading".last_run_4 = TRUE AND "Sensor_4" = TRUE THEN
           #Stop_sys := True;
       END_IF;
   // Kiểm tra xi lanh 5
   ELSIF #Alarm1_Bit13_cylinder5_Fault = TRUE THEN
       IF "Array_threading".array_threading_5[0] = 1 THEN
           "Array_threading".last_run_5 := True;
       END_IF;

       IF "Array_threading".last_run_5 = TRUE AND "Sensor_5" = TRUE THEN
           #Stop_sys := True;
       END_IF;
   END_IF;
END_REGION
END_FUNCTION

FUNCTION "Put_to_webserver" : Void   // FC5, LAD
{ S7_Optimized_Access := 'TRUE' }
VERSION : 0.1
   VAR_TEMP   // added for the SCL form of the ladder/FBD networks
      _w1 : Bool;
   END_VAR
BEGIN

REGION Network 1: state sensor
   // trang thai cam bien
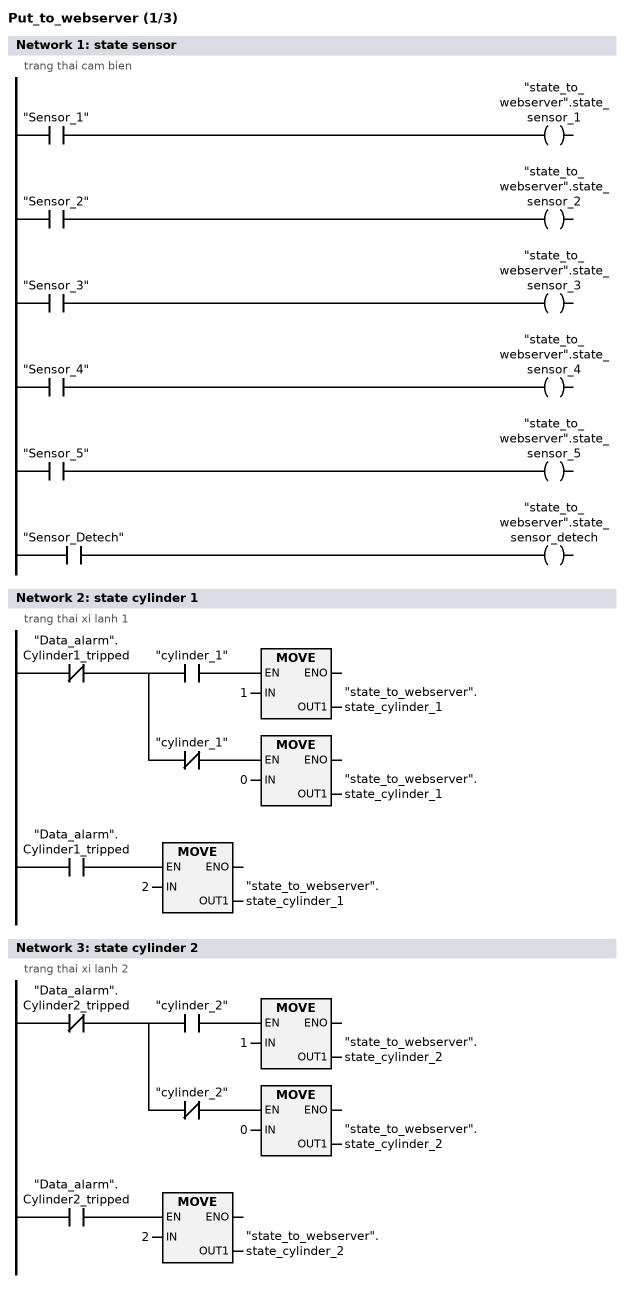
   RUNG wire#powerrail
      Contact( "Sensor_1" )
      Coil( "state_to_webserver".state_sensor_1 )
   END_RUNG
   RUNG wire#powerrail
      Contact( "Sensor_2" )
      Coil( "state_to_webserver".state_sensor_2 )
   END_RUNG
   RUNG wire#powerrail
      Contact( "Sensor_3" )
      Coil( "state_to_webserver".state_sensor_3 )
   END_RUNG
   RUNG wire#powerrail
      Contact( "Sensor_4" )
      Coil( "state_to_webserver".state_sensor_4 )
   END_RUNG
   RUNG wire#powerrail
      Contact( "Sensor_5" )
      Coil( "state_to_webserver".state_sensor_5 )
   END_RUNG
   RUNG wire#powerrail
      Contact( "Sensor_Detech" )
      Coil( "state_to_webserver".state_sensor_detech )
   END_RUNG
   // the same network as SCL:
   "state_to_webserver".state_sensor_1 := "Sensor_1";
   "state_to_webserver".state_sensor_2 := "Sensor_2";
   "state_to_webserver".state_sensor_3 := "Sensor_3";
   "state_to_webserver".state_sensor_4 := "Sensor_4";
   "state_to_webserver".state_sensor_5 := "Sensor_5";
   "state_to_webserver".state_sensor_detech := "Sensor_Detech";
END_REGION

REGION Network 2: state cylinder 1
   // trang thai xi lanh 1
   RUNG wire#powerrail
      I_Contact( "Data_alarm".Cylinder1_tripped )
      wire#w1
      Contact( "cylinder_1" )
      Move(in := 1, out1 => "state_to_webserver".state_cylinder_1)
   END_RUNG
   RUNG wire#w1
      I_Contact( "cylinder_1" )
      Move(in := 0, out1 => "state_to_webserver".state_cylinder_1)
   END_RUNG
   RUNG wire#powerrail
      Contact( "Data_alarm".Cylinder1_tripped )
      Move(in := 2, out1 => "state_to_webserver".state_cylinder_1)
   END_RUNG
   // the same network as SCL:
   #_w1 := NOT "Data_alarm".Cylinder1_tripped;
   IF #_w1 AND "cylinder_1" THEN "state_to_webserver".state_cylinder_1 := 1; END_IF;
   IF #_w1 AND NOT "cylinder_1" THEN "state_to_webserver".state_cylinder_1 := 0; END_IF;
   IF "Data_alarm".Cylinder1_tripped THEN "state_to_webserver".state_cylinder_1 := 2; END_IF;
END_REGION

REGION Network 3: state cylinder 2
   // trang thai xi lanh 2
   RUNG wire#powerrail
      I_Contact( "Data_alarm".Cylinder2_tripped )
      wire#w1
      Contact( "cylinder_2" )
      Move(in := 1, out1 => "state_to_webserver".state_cylinder_2)
   END_RUNG
   RUNG wire#w1
      I_Contact( "cylinder_2" )
      Move(in := 0, out1 => "state_to_webserver".state_cylinder_2)
   END_RUNG
   RUNG wire#powerrail
      Contact( "Data_alarm".Cylinder2_tripped )
      Move(in := 2, out1 => "state_to_webserver".state_cylinder_2)
   END_RUNG
   // the same network as SCL:
   #_w1 := NOT "Data_alarm".Cylinder2_tripped;
   IF #_w1 AND "cylinder_2" THEN "state_to_webserver".state_cylinder_2 := 1; END_IF;
   IF #_w1 AND NOT "cylinder_2" THEN "state_to_webserver".state_cylinder_2 := 0; END_IF;
   IF "Data_alarm".Cylinder2_tripped THEN "state_to_webserver".state_cylinder_2 := 2; END_IF;
END_REGION

REGION Network 4: state cylinder 3
   // trang thai xi lanh 3
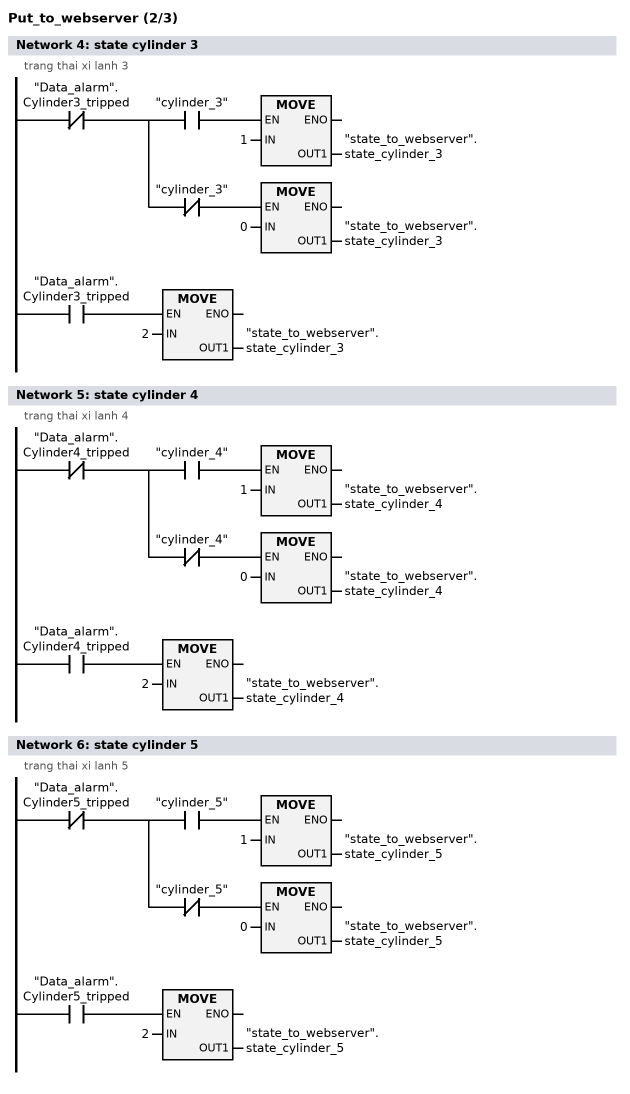
   RUNG wire#powerrail
      I_Contact( "Data_alarm".Cylinder3_tripped )
      wire#w1
      Contact( "cylinder_3" )
      Move(in := 1, out1 => "state_to_webserver".state_cylinder_3)
   END_RUNG
   RUNG wire#w1
      I_Contact( "cylinder_3" )
      Move(in := 0, out1 => "state_to_webserver".state_cylinder_3)
   END_RUNG
   RUNG wire#powerrail
      Contact( "Data_alarm".Cylinder3_tripped )
      Move(in := 2, out1 => "state_to_webserver".state_cylinder_3)
   END_RUNG
   // the same network as SCL:
   #_w1 := NOT "Data_alarm".Cylinder3_tripped;
   IF #_w1 AND "cylinder_3" THEN "state_to_webserver".state_cylinder_3 := 1; END_IF;
   IF #_w1 AND NOT "cylinder_3" THEN "state_to_webserver".state_cylinder_3 := 0; END_IF;
   IF "Data_alarm".Cylinder3_tripped THEN "state_to_webserver".state_cylinder_3 := 2; END_IF;
END_REGION

REGION Network 5: state cylinder 4
   // trang thai xi lanh 4
   RUNG wire#powerrail
      I_Contact( "Data_alarm".Cylinder4_tripped )
      wire#w1
      Contact( "cylinder_4" )
      Move(in := 1, out1 => "state_to_webserver".state_cylinder_4)
   END_RUNG
   RUNG wire#w1
      I_Contact( "cylinder_4" )
      Move(in := 0, out1 => "state_to_webserver".state_cylinder_4)
   END_RUNG
   RUNG wire#powerrail
      Contact( "Data_alarm".Cylinder4_tripped )
      Move(in := 2, out1 => "state_to_webserver".state_cylinder_4)
   END_RUNG
   // the same network as SCL:
   #_w1 := NOT "Data_alarm".Cylinder4_tripped;
   IF #_w1 AND "cylinder_4" THEN "state_to_webserver".state_cylinder_4 := 1; END_IF;
   IF #_w1 AND NOT "cylinder_4" THEN "state_to_webserver".state_cylinder_4 := 0; END_IF;
   IF "Data_alarm".Cylinder4_tripped THEN "state_to_webserver".state_cylinder_4 := 2; END_IF;
END_REGION

REGION Network 6: state cylinder 5
   // trang thai xi lanh 5
   RUNG wire#powerrail
      I_Contact( "Data_alarm".Cylinder5_tripped )
      wire#w1
      Contact( "cylinder_5" )
      Move(in := 1, out1 => "state_to_webserver".state_cylinder_5)
   END_RUNG
   RUNG wire#w1
      I_Contact( "cylinder_5" )
      Move(in := 0, out1 => "state_to_webserver".state_cylinder_5)
   END_RUNG
   RUNG wire#powerrail
      Contact( "Data_alarm".Cylinder5_tripped )
      Move(in := 2, out1 => "state_to_webserver".state_cylinder_5)
   END_RUNG
   // the same network as SCL:
   #_w1 := NOT "Data_alarm".Cylinder5_tripped;
   IF #_w1 AND "cylinder_5" THEN "state_to_webserver".state_cylinder_5 := 1; END_IF;
   IF #_w1 AND NOT "cylinder_5" THEN "state_to_webserver".state_cylinder_5 := 0; END_IF;
   IF "Data_alarm".Cylinder5_tripped THEN "state_to_webserver".state_cylinder_5 := 2; END_IF;
END_REGION

REGION Network 7: state motor conveyor
   // trang thai dong co bang tai
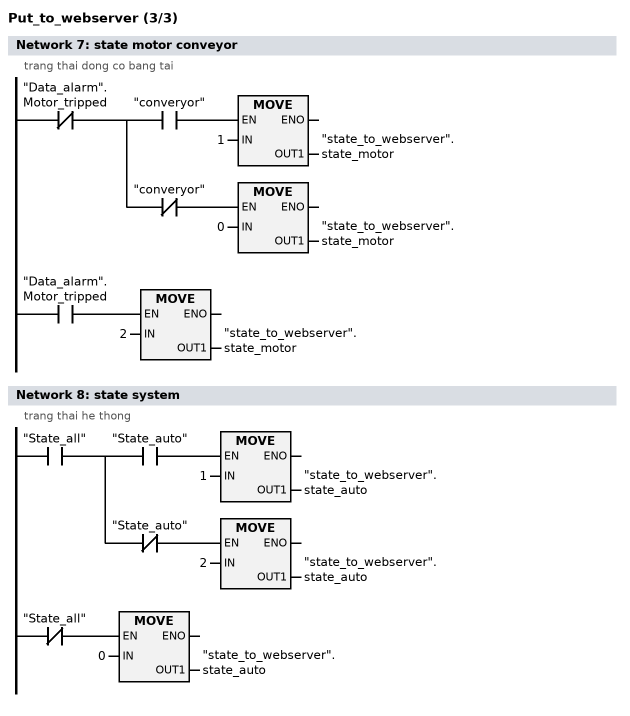
   RUNG wire#powerrail
      I_Contact( "Data_alarm".Motor_tripped )
      wire#w1
      Contact( "converyor" )
      Move(in := 1, out1 => "state_to_webserver".state_motor)
   END_RUNG
   RUNG wire#w1
      I_Contact( "converyor" )
      Move(in := 0, out1 => "state_to_webserver".state_motor)
   END_RUNG
   RUNG wire#powerrail
      Contact( "Data_alarm".Motor_tripped )
      Move(in := 2, out1 => "state_to_webserver".state_motor)
   END_RUNG
   // the same network as SCL:
   #_w1 := NOT "Data_alarm".Motor_tripped;
   IF #_w1 AND "converyor" THEN "state_to_webserver".state_motor := 1; END_IF;
   IF #_w1 AND NOT "converyor" THEN "state_to_webserver".state_motor := 0; END_IF;
   IF "Data_alarm".Motor_tripped THEN "state_to_webserver".state_motor := 2; END_IF;
END_REGION

REGION Network 8: state system
   // trang thai he thong
   RUNG wire#powerrail
      Contact( "State_all" )
      wire#w1
      Contact( "State_auto" )
      Move(in := 1, out1 => "state_to_webserver".state_auto)
   END_RUNG
   RUNG wire#w1
      I_Contact( "State_auto" )
      Move(in := 2, out1 => "state_to_webserver".state_auto)
   END_RUNG
   RUNG wire#powerrail
      I_Contact( "State_all" )
      Move(in := 0, out1 => "state_to_webserver".state_auto)
   END_RUNG
   // the same network as SCL:
   IF "State_all" AND "State_auto" THEN "state_to_webserver".state_auto := 1; END_IF;
   IF "State_all" AND NOT "State_auto" THEN "state_to_webserver".state_auto := 2; END_IF;
   IF NOT "State_all" THEN "state_to_webserver".state_auto := 0; END_IF;
END_REGION
END_FUNCTION

ORGANIZATION_BLOCK "Main"   // OB1, LAD, ProgramCycle
TITLE = "Main Program Sweep (Cycle)"
{ S7_Optimized_Access := 'TRUE' }
VERSION : 0.1
   VAR_TEMP   // added for the SCL form of the ladder/FBD networks
      _w1 : Bool;
   END_VAR
BEGIN

REGION Network 1: ON/OFF System
   // Bat tat toan bo he thong
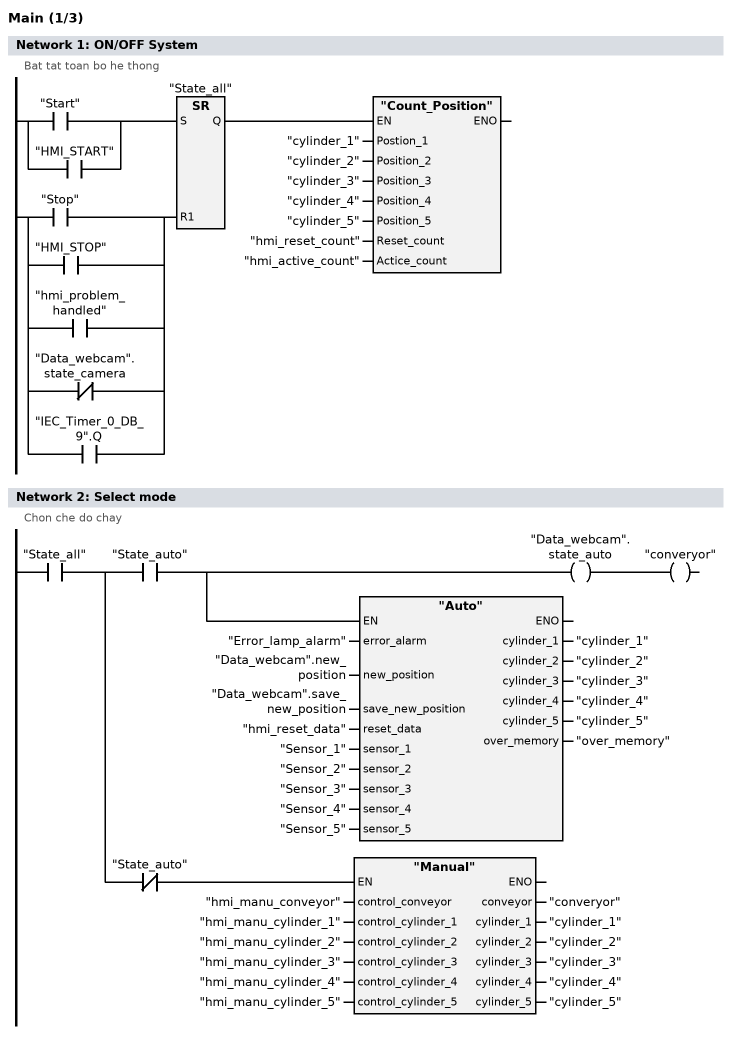
   RUNG wire#powerrail
      Contact( "Start" )
      wire#w1
      S_SR(operand := "State_all", r1 := wire#w2)
      "Count_Position"(Postion_1 := "cylinder_1", Position_2 := "cylinder_2", Position_3 := "cylinder_3", Position_4 := "cylinder_4", Position_5 := "cylinder_5", Reset_count := "hmi_reset_count", Actice_count := "hmi_active_count")
   END_RUNG
   RUNG wire#powerrail
      Contact( "HMI_START" )
   END_RUNG wire#w1
   RUNG wire#powerrail
      Contact( "Stop" )
   END_RUNG wire#w2
   RUNG wire#powerrail
      Contact( "HMI_STOP" )
   END_RUNG wire#w2
   RUNG wire#powerrail
      Contact( "hmi_problem_handled" )
   END_RUNG wire#w2
   RUNG wire#powerrail
      I_Contact( "Data_webcam".state_camera )
   END_RUNG wire#w2
   RUNG wire#powerrail
      Contact( "IEC_Timer_0_DB_9".Q )
   END_RUNG wire#w2
   // the same network as SCL:
   IF "Start" OR "HMI_START" THEN
       "State_all" := TRUE;   // SR flip-flop
   END_IF;
   IF "Stop" OR "HMI_STOP" OR "hmi_problem_handled" OR NOT "Data_webcam".state_camera OR "IEC_Timer_0_DB_9".Q THEN
       "State_all" := FALSE;
   END_IF;
   IF "State_all" THEN
       "Count_Position"(Postion_1 := "cylinder_1",
                        Position_2 := "cylinder_2",
                        Position_3 := "cylinder_3",
                        Position_4 := "cylinder_4",
                        Position_5 := "cylinder_5",
                        Reset_count := "hmi_reset_count",
                        Actice_count := "hmi_active_count");
   END_IF;
END_REGION

REGION Network 2: Select mode
   // Chon che do chay
   RUNG wire#powerrail
      Contact( "State_all" )
      wire#w1
      Contact( "State_auto" )
      wire#w2
      Coil( "Data_webcam".state_auto )
      Coil( "converyor" )
   END_RUNG
   RUNG wire#w2
      "Auto"(error_alarm := "Error_lamp_alarm", new_position := "Data_webcam".new_position, save_new_position := "Data_webcam".save_new_position, reset_data := "hmi_reset_data", sensor_1 := "Sensor_1", sensor_2 := "Sensor_2", sensor_3 := "Sensor_3", sensor_4 := "Sensor_4", sensor_5 := "Sensor_5", cylinder_1 => "cylinder_1", cylinder_2 => "cylinder_2", cylinder_3 => "cylinder_3", cylinder_4 => "cylinder_4", cylinder_5 => "cylinder_5", over_memory => "over_memory")
   END_RUNG
   RUNG wire#w1
      I_Contact( "State_auto" )
      "Manual"(control_conveyor := "hmi_manu_conveyor", control_cylinder_1 := "hmi_manu_cylinder_1", control_cylinder_2 := "hmi_manu_cylinder_2", control_cylinder_3 := "hmi_manu_cylinder_3", control_cylinder_4 := "hmi_manu_cylinder_4", control_cylinder_5 := "hmi_manu_cylinder_5", conveyor => "converyor", cylinder_1 => "cylinder_1", cylinder_2 => "cylinder_2", cylinder_3 => "cylinder_3", cylinder_4 => "cylinder_4", cylinder_5 => "cylinder_5")
   END_RUNG
   // the same network as SCL:
   "Data_webcam".state_auto := "State_all" AND "State_auto";
   "converyor" := "Data_webcam".state_auto;
   #_w1 := "State_all";
   IF "Data_webcam".state_auto THEN
       "Auto"(error_alarm := "Error_lamp_alarm",
              new_position := "Data_webcam".new_position,
              save_new_position := "Data_webcam".save_new_position,
              reset_data := "hmi_reset_data",
              sensor_1 := "Sensor_1",
              sensor_2 := "Sensor_2",
              sensor_3 := "Sensor_3",
              sensor_4 := "Sensor_4",
              sensor_5 := "Sensor_5",
              cylinder_1 => "cylinder_1",
              cylinder_2 => "cylinder_2",
              cylinder_3 => "cylinder_3",
              cylinder_4 => "cylinder_4",
              cylinder_5 => "cylinder_5",
              over_memory => "over_memory");
   END_IF;
   IF #_w1 AND NOT "State_auto" THEN
       "Manual"(control_conveyor := "hmi_manu_conveyor",
                control_cylinder_1 := "hmi_manu_cylinder_1",
                control_cylinder_2 := "hmi_manu_cylinder_2",
                control_cylinder_3 := "hmi_manu_cylinder_3",
                control_cylinder_4 := "hmi_manu_cylinder_4",
                control_cylinder_5 := "hmi_manu_cylinder_5",
                conveyor => "converyor",
                cylinder_1 => "cylinder_1",
                cylinder_2 => "cylinder_2",
                cylinder_3 => "cylinder_3",
                cylinder_4 => "cylinder_4",
                cylinder_5 => "cylinder_5");
   END_IF;
END_REGION

REGION Network 3: connect to function
   // ket noi cac function con lai
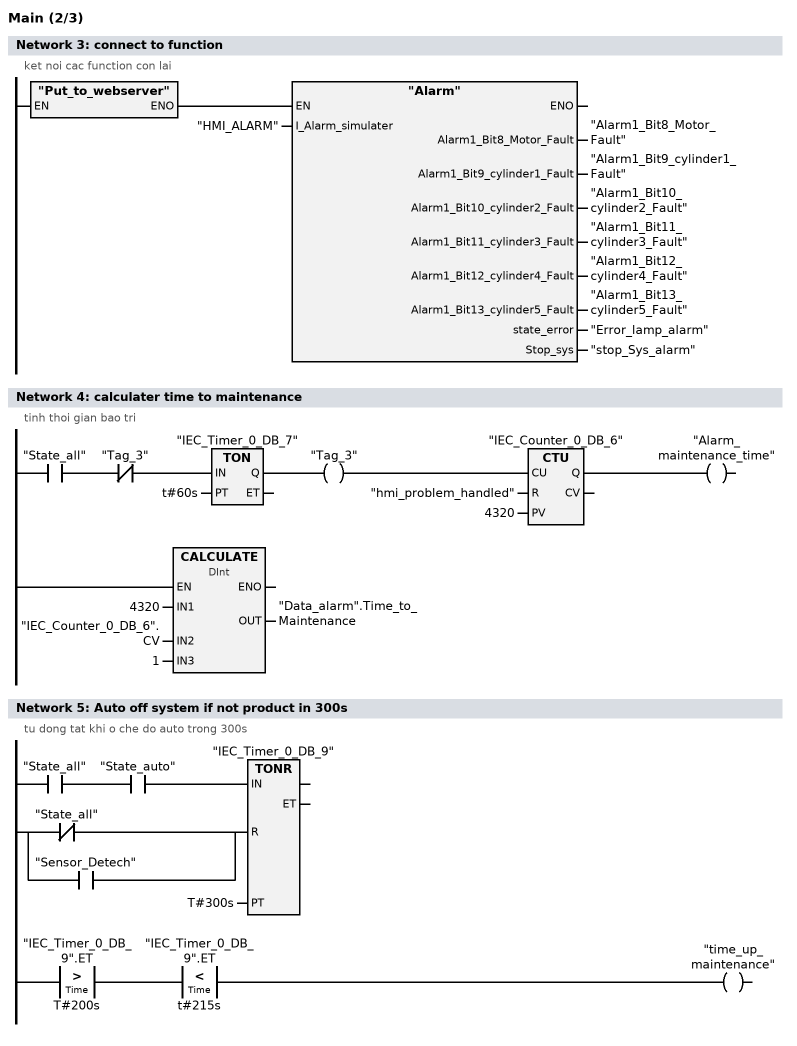
   RUNG wire#powerrail
      "Put_to_webserver"()
      "Alarm"(I_Alarm_simulater := "HMI_ALARM", Alarm1_Bit8_Motor_Fault => "Alarm1_Bit8_Motor_Fault", Alarm1_Bit9_cylinder1_Fault => "Alarm1_Bit9_cylinder1_Fault", Alarm1_Bit10_cylinder2_Fault => "Alarm1_Bit10_cylinder2_Fault", Alarm1_Bit11_cylinder3_Fault => "Alarm1_Bit11_cylinder3_Fault", Alarm1_Bit12_cylinder4_Fault => "Alarm1_Bit12_cylinder4_Fault", Alarm1_Bit13_cylinder5_Fault => "Alarm1_Bit13_cylinder5_Fault", state_error => "Error_lamp_alarm", Stop_sys => "stop_Sys_alarm")
   END_RUNG
   // the same network as SCL:
   "Put_to_webserver"(ENO => #_w1);
   IF #_w1 THEN
       "Alarm"(I_Alarm_simulater := "HMI_ALARM",
               Alarm1_Bit8_Motor_Fault => "Alarm1_Bit8_Motor_Fault",
               Alarm1_Bit9_cylinder1_Fault => "Alarm1_Bit9_cylinder1_Fault",
               Alarm1_Bit10_cylinder2_Fault => "Alarm1_Bit10_cylinder2_Fault",
               Alarm1_Bit11_cylinder3_Fault => "Alarm1_Bit11_cylinder3_Fault",
               Alarm1_Bit12_cylinder4_Fault => "Alarm1_Bit12_cylinder4_Fault",
               Alarm1_Bit13_cylinder5_Fault => "Alarm1_Bit13_cylinder5_Fault",
               state_error => "Error_lamp_alarm",
               Stop_sys => "stop_Sys_alarm");
   END_IF;
END_REGION

REGION Network 4: calculater time to maintenance
   // tinh thoi gian bao tri
   "IEC_Timer_0_DB_7".TON(IN := "State_all" AND NOT "Tag_3", PT := t#60s);
   "Tag_3" := "IEC_Timer_0_DB_7".Q;
   "IEC_Counter_0_DB_6".CTU(CU := "IEC_Timer_0_DB_7".Q, R := "hmi_problem_handled", PV := 4320);
   "Alarm_maintenance_time" := "IEC_Counter_0_DB_6".Q;
   "Data_alarm".Time_to_Maintenance := (4320 - "IEC_Counter_0_DB_6".CV)*1;
END_REGION

REGION Network 5: Auto off system if not product in 300s
   // tu dong tat khi o che do auto trong 300s
   "IEC_Timer_0_DB_9".TONR(IN := "State_all" AND "State_auto",
                           R := NOT "State_all" OR "Sensor_Detech",
                           PT := T#300s);
   "time_up_maintenance" := ("IEC_Timer_0_DB_9".ET > T#200s) AND ("IEC_Timer_0_DB_9".ET < t#215s);
END_REGION

REGION Network 6: Alarm lamp
   // den canh bao
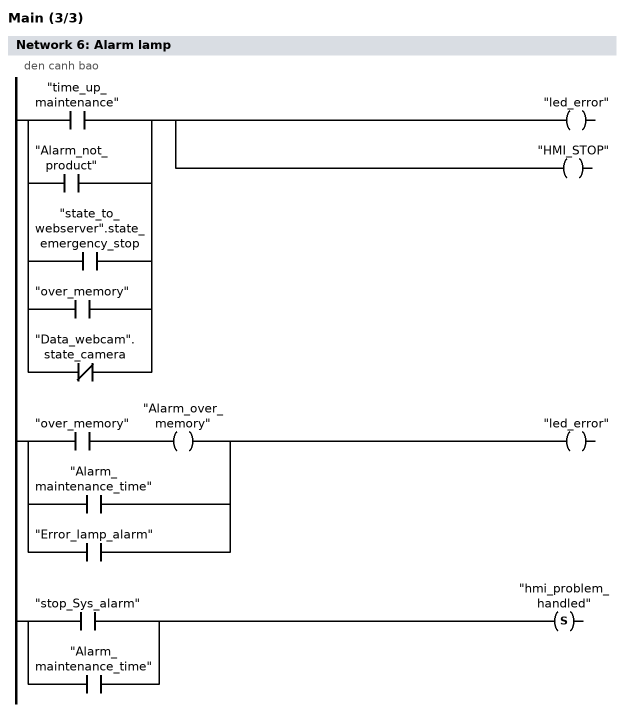
   RUNG wire#powerrail
      Contact( "time_up_maintenance" )
      wire#w1
      Coil( "led_error" )
   END_RUNG
   RUNG wire#powerrail
      Contact( "Alarm_not_product" )
   END_RUNG wire#w1
   RUNG wire#powerrail
      Contact( "state_to_webserver".state_emergency_stop )
   END_RUNG wire#w1
   RUNG wire#powerrail
      Contact( "over_memory" )
   END_RUNG wire#w1
   RUNG wire#powerrail
      I_Contact( "Data_webcam".state_camera )
   END_RUNG wire#w1
   RUNG wire#w1
      Coil( "HMI_STOP" )
   END_RUNG
   RUNG wire#powerrail
      Contact( "over_memory" )
      Coil( "Alarm_over_memory" )
      wire#w2
      Coil( "led_error" )
   END_RUNG
   RUNG wire#powerrail
      Contact( "Alarm_maintenance_time" )
   END_RUNG wire#w2
   RUNG wire#powerrail
      Contact( "Error_lamp_alarm" )
   END_RUNG wire#w2
   RUNG wire#powerrail
      Contact( "stop_Sys_alarm" )
      wire#w3
      S_Coil( "hmi_problem_handled" )
   END_RUNG
   RUNG wire#powerrail
      Contact( "Alarm_maintenance_time" )
   END_RUNG wire#w3
   // the same network as SCL:
   "led_error" := "time_up_maintenance" OR "Alarm_not_product" OR "state_to_webserver".state_emergency_stop OR "over_memory" OR NOT "Data_webcam".state_camera;
   "HMI_STOP" := "led_error";
   "Alarm_over_memory" := "over_memory";
   "led_error" := "over_memory" OR "Alarm_maintenance_time" OR "Error_lamp_alarm";
   IF "stop_Sys_alarm" OR "Alarm_maintenance_time" THEN "hmi_problem_handled" := TRUE; END_IF;
END_REGION
END_ORGANIZATION_BLOCK

(* ===== HMI "HMI_RT_1" =====
system functions are stored by id; their names below are inferred from use
connection "HMI_Connection_1": ETHERNET, SMART_S7_1200_OMS

HMI tags "Default tag table"
   "State_auto" : Bool = PLC State_auto AT %M10.1, 1 s
   "Start" : Bool = PLC Start AT %I0.0, 1 s
   "Stop" : Bool = PLC Stop AT %I0.1, 1 s
   "converyor" : Bool = PLC converyor AT %Q1.0, 1 s
   "cylinder_1" : Bool = PLC cylinder_1 AT %Q0.1, 1 s
   "cylinder_2" : Bool = PLC cylinder_2 AT %Q1.1, 1 s
   "cylinder_3" : Bool = PLC cylinder_3 AT %Q0.3, 1 s
   "cylinder_4" : Bool = PLC cylinder_4 AT %Q0.4, 1 s
   "cylinder_5" : Bool = PLC cylinder_5 AT %Q0.5, 1 s
   "m_active_count" : Bool = PLC hmi_active_count AT %M11.0, 1 s
   "m_manu_cylinder_1" : Bool = PLC hmi_manu_cylinder_1 AT %M10.3, 1 s
   "m_manu_cylinder_2" : Bool = PLC hmi_manu_cylinder_2 AT %M10.4, 1 s
   "m_manu_cylinder_3" : Bool = PLC hmi_manu_cylinder_3 AT %M10.5, 1 s
   "m_manu_cylinder_4" : Bool = PLC hmi_manu_cylinder_4 AT %M10.6, 1 s
   "m_manu_cylinder_5" : Bool = PLC hmi_manu_cylinder_5 AT %M10.7, 1 s
   "Alarm1_Bit0" : Bool = PLC Alarm1_Bit0 AT %M21.0, 1 s
   "Alarm1" : Word = PLC Alarm1 AT %MW20, 1 s
   "HMI_ALARM" : Bool = PLC HMI_ALARM AT %M11.1, 1 s
   "m_manual_conveyor" : Bool = PLC hmi_manu_conveyor AT %M10.2, 1 s
   "HMI_START" : Bool = PLC HMI_START AT %M11.2, 1 s
   "HMI_STOP" : Bool = PLC HMI_STOP AT %M11.3, 1 s
   "Data_count_Position_Adress_1" : Real = PLC Data_count_Position.Adress_1 AT %DB8.DBD0, 1 s
   "Data_count_Position_Adress_2" : Real = PLC Data_count_Position.Adress_2 AT %DB8.DBD4, 1 s
   "Data_count_Position_Adress_3" : Real = PLC Data_count_Position.Adress_3 AT %DB8.DBD8, 1 s
   "Data_count_Position_Adress_4" : Real = PLC Data_count_Position.Adress_4 AT %DB8.DBD12, 1 s
   "Data_count_Position_Adress_5" : Real = PLC Data_count_Position.Adress_5 AT %DB8.DBD16, 1 s
   "Data_count_Position_Adress_6" : Real = PLC Data_count_Position.Adress_6 AT %DB8.DBD20, 1 s
   "Sensor_1" : Bool = PLC Sensor_1 AT %I0.3, 1 s
   "Sensor_2" : Bool = PLC Sensor_2 AT %I0.4, 1 s
   "Sensor_3" : Bool = PLC Sensor_3 AT %I0.5, 1 s
   "Sensor_4" : Bool = PLC Sensor_4 AT %I0.6, 1 s
   "Sensor_5" : Bool = PLC Sensor_5 AT %I0.7, 1 s
   "led_error" : Bool = PLC led_error AT %Q0.6, 1 s
   "Actice_count" : Bool = PLC hmi_active_count AT %M11.0, 1 s
   "State_all" : Bool = PLC State_all AT %M10.0, 1 s
   "Sim_motor_tripped" : Bool = PLC Sim_motor_tripped AT %M52.0, 1 s
   "Sim_cylinder1_tripped" : Bool = PLC Sim_cylinder1_tripped AT %M52.1, 1 s
   "Sim_cylinder3_tripped" : Bool = PLC Sim_cylinder3_tripped AT %M52.3, 1 s
   "Sim_cylinder4_tripped" : Bool = PLC Sim_cylinder4_tripped AT %M52.4, 1 s
   "Sim_cylinder5_tripped" : Bool = PLC Sim_cylinder5_tripped AT %M52.5, 1 s
   "Sim_cylinder2_tripped" : Bool = PLC Sim_cylinder2_tripped AT %M52.2, 1 s
   "hmi_problem_handled" : Bool = PLC hmi_problem_handled AT %M11.5, 1 s
   "Sensor_Detech" : Bool = PLC Sensor_Detech AT %I0.2, 1 s
   "Data_alarm_Time_to_Maintenance" : DInt = PLC Data_alarm.Time_to_Maintenance AT %DB17.DBD2, 1 s
   "hmi_reset_count" : Bool = PLC hmi_reset_count AT %M11.4, 1 s
   "hmi_reset_data" : Bool = PLC hmi_reset_data AT %M11.6, 1 s
   "state_to_webserver_state_emergency_stop" : Bool = PLC state_to_webserver.state_emergency_stop AT %DB22.DBX0.6, 1 s
   "Data_webcam_state_camera" : Bool = PLC Data_webcam.state_camera AT %DB7.DBX2.1, 1 s

HMI tags "INTERNAL TAGS"
   "Screen_id" : Int AT %DB1.DBW0

HMI tags "User_name"
   "Username" : WString[50], internal

discrete alarms
   1: 'Động cơ bị sự cố', class Errors, trigger "Alarm1" bit 8
   2: 'Xi lanh 1 bị sự cố', class Errors, trigger "Alarm1" bit 9
   3: 'Xi lanh 2 bị sự cố', class Errors, trigger "Alarm1" bit 10
   4: 'Xi lanh 3 bị sự cố', class Errors, trigger "Alarm1" bit 11
   5: 'Xi lanh 4 bị sự cố', class Errors, trigger "Alarm1" bit 12
   6: 'Xi lanh 5 bị sự cố', class Errors, trigger "Alarm1" bit 13
   7: 'Tới thời gian bảo trì', class Warnings, trigger "Alarm1" bit 7
   8: 'Mất kết nối với Camera', class Errors, trigger "Alarm1" bit 6
   9: 'Dừng khẩn cấp từ webserver', class Errors, trigger "Alarm1" bit 5
   10: 'Vượt quá dữ liệu phân loại cho phép , vui lòng đợi', class Warnings, trigger "Alarm1" bit 4

graphic list "Motor": 0 'Graphic_2'; 1 'Graphic_3'

graphic list "bang_tai": 0..1 'Graphic_4'; 1 'Graphic_5'

graphic list "hop": 0 'Graphic_9'

graphic list "cambien": 0..1 'Graphic_15'; 1 'Graphic_16'

Template "Template_1" 800x480
   TextField "Text field_1" at -4202,109 size 16x23; Text 'Text'
   GraphicView "Graphic view_1" at 2,0 size 96x90; Picture "download"
   TextField "Text field_2" at 141,9 size 227x27; Text 'SIEMENS HMI COURSE'
   TextField "Text field_3" at 130,47 size 259x25; Text 'instructor: Vĩnh hiển and Hữu Đạt'
   Button "Button_1" at 431,0 size 92x90; TextOff 'HOME'
      on Press: ActivateScreen("Screen_home", 0); SetTag("Screen_id", 0)
      Appearance <- "Screen_id"
   Button "Button_2" at 523,0 size 92x90; TextOff 'SETTING'; Authorization "Operate"
      on Press: ActivateScreen("Screen_Setting", 0); SetTag("Screen_id", 1)
      Appearance <- "Screen_id"
   Button "Button_3" at 615,0 size 92x90; TextOff 'ALARM'; Authorization "Operate"
      on Press: ActivateScreen("Screen_ALARM", 0); SetTag("Screen_id", 2)
      Appearance <- "Screen_id"
   Button "Button_4" at 707,0 size 92x90; TextOff 'ADMIN'; Authorization "User administration"
      on Press: ActivateScreen("Screen_ADMIN", 0); SetTag("Screen_id", 3)
      Appearance <- "Screen_id"
   Softkey "Softkey_F1" at 0,0 size 0x0
      on KeyDown: ActivateScreen("Screen_Setting", 0)
   Softkey "Softkey_F2" at 0,0 size 0x0
      on KeyDown: ActivateScreen("AUTO", 0)
   Softkey "Softkey_F3" at 0,0 size 0x0
      on KeyDown: ActivateScreen("MANU", 0)
   Softkey "Softkey_F4" at 0,0 size 0x0
      on KeyDown: ActivateScreen("Screen_ALARM", 0)
   Softkey "Softkey_F8" at 0,0 size 0x0
      on KeyDown: ActivateScreen("Test_IO", 0)

screen "Screen_home" 800x480, template "Template_1"
   TextField "Text field_1" at 296,179 size 193x25; Text 'Current problem table'
   AlarmView "Alarm view_1" at 4,207 size 789x266
   Button "Button_1" at 13,102 size 93x28; TextOff 'Login'
      on Press: function_a2a04561()
   Button "Button_2" at 12,141 size 93x28; TextOff 'Logout'
      on Press: function_f23ef4c9()
   IOField "I/O field_1" at 149,131 size 160x32; FormatPattern ??????????????????????????????????????????????????
      ProcessValue <- "Username"
   TextField "Text field_2" at 147,95 size 98x23; Text 'User login :'
   Circle "Circle_1" at 674,121 size 48x48
      Appearance <- "led_error"
   TextField "Text field_3" at 620,94 size 165x23; Text 'Error indicator light'
   Button "Button_3" at 392,131 size 202x32; TextOff 'The problem has been handled'; Authorization "User administration"
      on Click: ResetBit("hmi_problem_handled")
      Appearance <- "hmi_problem_handled"
      Visibility <- "hmi_problem_handled"

screen "Screen_Setting" 800x480, template "Template_1"
   GraphicView "Graphic view_1" at 205,90 size 594x388; Picture "anh"
   Switch "Switch_1" at 56,225 size 122x32; CaptionText 'Switch'; TextOff 'MANU'; TextOn 'AUTO'; Authorization "Operate"
      ProcessValue <- "State_auto"
   TextField "Text field_1" at 54,190 size 121x23; Text 'Select mode :'
   Button "Button_1" at 7,282 size 96x32; TextOff 'AUTO'; Authorization "Operate"
      on Press: ActivateScreen("AUTO", 0); SetTag("Screen_id", 4)
      Appearance <- "State_auto"
   Button "Button_2" at 126,282 size 96x32; TextOff 'MANU'; Authorization "Operate"
      on Press: ActivateScreen("MANU", 0); SetTag("Screen_id", 5)
      Appearance <- "State_auto"
   Button "Button_3" at 10,138 size 98x34; TextOff 'START'; Authorization "Operate"
      on Release: ResetBit("HMI_START")
      on Press: SetBit("HMI_START")
      Appearance <- "State_all"
   Button "Button_4" at 131,138 size 93x34; TextOff 'STOP'; Authorization "Operate"
      on Release: ResetBit("HMI_STOP")
      on Press: SetBit("HMI_STOP")
      Appearance <- "State_all"
   TextField "Text field_2" at 14,347 size 193x22; Text 'Count classified products'
   Switch "Switch_2" at 84,380 size 64x32; CaptionText 'Switch'; TextOff 'OFF'; TextOn 'ON'; Authorization "User administration"
      ProcessValue <- "Actice_count"
   Button "Button_5" at 60,427 size 116x32; TextOff 'Reset Counter'; Authorization "User administration"
      on Press: SetBit("hmi_reset_count")
      on Release: ResetBit("hmi_reset_count")
   TextField "Text field_3" at 267,122 size 188x23; Text 'Time to Maintenance :'
   IOField "I/O field_1" at 459,119 size 76x32; FormatPattern 99999
      ProcessValue <- "Data_alarm_Time_to_Maintenance"
   TextField "Text field_4" at 537,123 size 61x23; Text 'Minute'

screen "Screen_ADMIN" 800x480, template "Template_1"
   UserView "User view_1" at 0,128 size 799x351
   TextField "Text field_1" at 364,99 size 72x23; Text 'User list'

screen "Screen_ALARM" 800x480, template "Template_1"
   TextField "Text field_1" at 58,112 size 16x23; Text 'Text'
   TextField "Text field_2" at 77,112 size 73x23; Text 'Problem'
   Button "Button_2" at 29,207 size 160x36; TextOff 'Conveyor Tripped'; Authorization "User administration"
      on Press: InvertBit("Sim_motor_tripped")
      Appearance <- "Sim_motor_tripped"
   Button "Button_3" at 29,251 size 160x36; TextOff 'Cylinder 1 Tripped'; Authorization "User administration"
      on Press: InvertBit("Sim_cylinder1_tripped")
      Appearance <- "Sim_cylinder1_tripped"
   Button "Button_4" at 29,296 size 160x36; TextOff 'Cylinder 2 Tripped'; Authorization "User administration"
      on Press: InvertBit("Sim_cylinder2_tripped")
      Appearance <- "Sim_cylinder2_tripped"
   Button "Button_5" at 29,386 size 160x36; TextOff 'Cylinder 4 Tripped'; Authorization "User administration"
      on Press: InvertBit("Sim_cylinder4_tripped")
      Appearance <- "Sim_cylinder4_tripped"
   Button "Button_6" at 29,341 size 160x36; TextOff 'Cylinder 3 Tripped'; Authorization "User administration"
      on Press: InvertBit("Sim_cylinder3_tripped")
      Appearance <- "Sim_cylinder3_tripped"
   Button "Button_7" at 29,431 size 160x36; TextOff 'Cylinder 5 Tripped'; Authorization "User administration"
      on Press: InvertBit("Sim_cylinder5_tripped")
      Appearance <- "Sim_cylinder5_tripped"
   AlarmView "Alarm view_1" at 214,87 size 582x390
   Switch "Switch_1" at 137,153 size 64x32; CaptionText 'Switch'; TextOff 'OFF'; TextOn 'ON'; Authorization "User administration"
      ProcessValue <- "HMI_ALARM"
   TextField "Text field_3" at 28,156 size 95x23; Text 'Simulater :'

screen "AUTO" 800x480, template "Template_1"
   GraphicIOField "Graphic I/O field_2" at 218,318 size 307x38; PictureList "bang_tai"
      ProcessValue <- "converyor"
   GraphicIOField "Graphic I/O field_5" at 476,317 size 323x38; PictureList "bang_tai"
      ProcessValue <- "converyor"
   GraphicView "Graphic view_1" at 360,203 size 22x94; Picture "Graphic_13"
      Visibility <- "cylinder_1"
   TextField "Text field_1" at 48,183 size 105x23; Text 'MODE AUTO'
   Rectangle "Rectangle_3" at 7,255 size 90x35
      Appearance <- "converyor"
   Rectangle "Rectangle_4" at 116,255 size 90x35
      Appearance <- "cylinder_1"
   Rectangle "Rectangle_5" at 116,312 size 90x35
      Appearance <- "cylinder_3"
   Rectangle "Rectangle_6" at 116,368 size 90x35
      Appearance <- "cylinder_5"
   Rectangle "Rectangle_7" at 7,312 size 90x35
      Appearance <- "cylinder_2"
   Rectangle "Rectangle_8" at 7,366 size 90x35
      Appearance <- "cylinder_4"
   TextField "Text field_2" at 24,261 size 58x23; Text 'Motor'
   TextField "Text field_3" at 117,261 size 87x23; Text 'Cylinder 1'
   TextField "Text field_4" at 8,316 size 87x23; Text 'Cylinder 2'
   TextField "Text field_5" at 117,317 size 87x23; Text 'Cylinder 3'
   TextField "Text field_6" at 8,376 size 87x23; Text 'Cylinder 4'
   TextField "Text field_7" at 117,374 size 87x23; Text 'Cylinder 5'
   GraphicIOField "Graphic I/O field_1" at 227,361 size 64x41; PictureList "Motor"
      ProcessValue <- "converyor"
   GraphicIOField "Graphic I/O field_11" at 334,375 size 80x48; PictureList "hop"
   GraphicIOField "Graphic I/O field_12" at 427,375 size 80x48; PictureList "hop"
   GraphicIOField "Graphic I/O field_13" at 520,375 size 80x48; PictureList "hop"
   GraphicIOField "Graphic I/O field_14" at 613,375 size 80x48; PictureList "hop"
   GraphicIOField "Graphic I/O field_15" at 707,375 size 80x48; PictureList "hop"
   IOField "I/O field_2" at 344,435 size 60x30; FormatPattern 9999
      ProcessValue <- "Data_count_Position_Adress_1"
   IOField "I/O field_3" at 437,435 size 60x30; FormatPattern 9999
      ProcessValue <- "Data_count_Position_Adress_2"
   IOField "I/O field_4" at 530,435 size 60x30; FormatPattern 9999
      ProcessValue <- "Data_count_Position_Adress_3"
   IOField "I/O field_5" at 623,435 size 60x30; FormatPattern 9999
      ProcessValue <- "Data_count_Position_Adress_4"
   IOField "I/O field_6" at 716,435 size 60x30; FormatPattern 9999
      ProcessValue <- "Data_count_Position_Adress_5"
   GraphicIOField "Graphic I/O field_16" at 273,264 size 25x48; PictureList "cambien"
      ProcessValue <- "Sensor_Detech"
   GraphicIOField "Graphic I/O field_17" at 386,214 size 25x48; PictureList "cambien"
      ProcessValue <- "Sensor_1"
   GraphicIOField "Graphic I/O field_18" at 473,214 size 25x48; PictureList "cambien"
      ProcessValue <- "Sensor_2"
   GraphicIOField "Graphic I/O field_19" at 569,214 size 25x48; PictureList "cambien"
      ProcessValue <- "Sensor_3"
   GraphicIOField "Graphic I/O field_20" at 667,214 size 25x48; PictureList "cambien"
      ProcessValue <- "Sensor_4"
   GraphicIOField "Graphic I/O field_21" at 761,214 size 25x48; PictureList "cambien"
      ProcessValue <- "Sensor_5"
   Circle "Circle_1" at 681,124 size 48x48
      Appearance <- "led_error"
   TextField "Text field_8" at 627,97 size 165x23; Text 'Error indicator light'
   GraphicView "Graphic view_4" at 361,203 size 22x60; Picture "Graphic_14"
      Visibility <- "cylinder_1"
   GraphicView "Graphic view_2" at 449,203 size 22x94; Picture "Graphic_13"
      Visibility <- "cylinder_2"
   GraphicView "Graphic view_3" at 450,203 size 22x60; Picture "Graphic_14"
      Visibility <- "cylinder_2"
   GraphicView "Graphic view_5" at 548,203 size 22x94; Picture "Graphic_13"
      Visibility <- "cylinder_3"
   GraphicView "Graphic view_6" at 549,203 size 22x60; Picture "Graphic_14"
      Visibility <- "cylinder_3"
   GraphicView "Graphic view_7" at 641,203 size 22x94; Picture "Graphic_13"
      Visibility <- "cylinder_4"
   GraphicView "Graphic view_8" at 642,203 size 22x60; Picture "Graphic_14"
      Visibility <- "cylinder_4"
   GraphicView "Graphic view_9" at 738,203 size 22x94; Picture "Graphic_13"
      Visibility <- "cylinder_5"
   GraphicView "Graphic view_10" at 739,203 size 22x60; Picture "Graphic_14"
      Visibility <- "cylinder_5"
   Group "Group" at 218,317 size 581x39; PictureList "bang_tai"
   TextField "Text field_9" at 360,176 size 69x23; Text 'Group 1'
   TextField "Text field_10" at 451,176 size 69x23; Text 'Group 2'
   TextField "Text field_11" at 543,176 size 69x23; Text 'Group 3'
   TextField "Text field_12" at 635,176 size 69x23; Text 'Group 4'
   TextField "Text field_13" at 727,176 size 69x23; Text 'Group 5'
   Button "Button_1" at 238,190 size 96x32; TextOff 'Reset data'
      on Press: SetBit("hmi_reset_data")
      on Release: ResetBit("hmi_reset_data")
   Circle "Circle_2" at 503,124 size 48x48
      Appearance <- "state_to_webserver_state_emergency_stop"
   TextField "Text field_14" at 429,97 size 190x23; Text 'Lock run by Webserver'
   Circle "Circle_3" at 287,124 size 48x48
      Appearance <- "Data_webcam_state_camera"
   TextField "Text field_15" at 231,97 size 177x23; Text 'Connect with camera'

screen "MANU" 800x480, template "Template_1"
   TextField "Text field_1" at 37,104 size 128x22; Text 'MODE MANUAL:'
   Button "Button_1" at 12,147 size 75x36; TextOff 'Motor'; Authorization "Operate"
      on Press: InvertBit("m_manual_conveyor")
   Rectangle "Rectangle_1" at 99,147 size 100x36
      Appearance <- "converyor"
   TextField "Text field_2" at 122,153 size 53x23; Text 'Motor'
   Button "Button_2" at 12,202 size 75x36; TextOff 'Cylinder 1'; Authorization "Operate"
      on Press: InvertBit("m_manu_cylinder_1")
   Rectangle "Rectangle_3" at 99,202 size 100x36
      Appearance <- "cylinder_1"
   TextField "Text field_3" at 106,210 size 87x23; Text 'Cylinder 1'
   Button "Button_3" at 12,257 size 75x36; TextOff 'Cylinder 2'; Authorization "Operate"
      on Press: InvertBit("m_manu_cylinder_2")
   Rectangle "Rectangle_4" at 99,257 size 100x36
      Appearance <- "cylinder_2"
   TextField "Text field_4" at 106,267 size 87x23; Text 'Cylinder 2'
   Button "Button_4" at 12,312 size 75x36; TextOff 'Cylinder 3'; Authorization "Operate"
      on Press: InvertBit("m_manu_cylinder_3")
   Rectangle "Rectangle_5" at 100,312 size 100x36
      Appearance <- "cylinder_3"
   TextField "Text field_5" at 106,320 size 87x23; Text 'Cylinder 3'
   Button "Button_5" at 12,367 size 75x36; TextOff 'Cylinder 4'; Authorization "Operate"
      on Press: InvertBit("m_manu_cylinder_4")
   Rectangle "Rectangle_6" at 100,367 size 100x36
      Appearance <- "cylinder_4"
   TextField "Text field_6" at 106,376 size 87x23; Text 'Cylinder 4'
   Button "Button_6" at 12,423 size 75x36; TextOff 'Cylinder 5'; Authorization "Operate"
      on Press: InvertBit("m_manu_cylinder_5")
   Rectangle "Rectangle_7" at 100,423 size 100x36
      Appearance <- "cylinder_5"
   TextField "Text field_7" at 106,430 size 87x23; Text 'Cylinder 5'
   GraphicIOField "Graphic I/O field_1" at 227,361 size 64x41; PictureList "Motor"
      ProcessValue <- "converyor"
   GraphicIOField "Graphic I/O field_11" at 334,375 size 80x48; PictureList "hop"
   GraphicIOField "Graphic I/O field_12" at 427,375 size 80x48; PictureList "hop"
   GraphicIOField "Graphic I/O field_13" at 520,375 size 80x48; PictureList "hop"
   GraphicIOField "Graphic I/O field_14" at 613,375 size 80x48; PictureList "hop"
   IOField "I/O field_2" at 344,435 size 60x30; FormatPattern 9999
      ProcessValue <- "Data_count_Position_Adress_1"
   IOField "I/O field_3" at 437,435 size 60x30; FormatPattern 9999
      ProcessValue <- "Data_count_Position_Adress_2"
   IOField "I/O field_4" at 530,435 size 60x30; FormatPattern 9999
      ProcessValue <- "Data_count_Position_Adress_3"
   IOField "I/O field_5" at 623,435 size 60x30; FormatPattern 9999
      ProcessValue <- "Data_count_Position_Adress_4"
   IOField "I/O field_6" at 716,435 size 60x30; FormatPattern 9999
      ProcessValue <- "Data_count_Position_Adress_5"
   Group "Group" at 218,317 size 581x39; PictureList "bang_tai"
   GraphicIOField "Graphic I/O field_15" at 707,375 size 80x48; PictureList "hop"
   GraphicView "Graphic view_1" at 360,203 size 22x94; Picture "Graphic_13"
      Visibility <- "cylinder_1"
   GraphicIOField "Graphic I/O field_16" at 273,264 size 25x48; PictureList "cambien"
      ProcessValue <- "Sensor_Detech"
   GraphicIOField "Graphic I/O field_17" at 386,214 size 25x48; PictureList "cambien"
      ProcessValue <- "Sensor_1"
   GraphicIOField "Graphic I/O field_18" at 473,214 size 25x48; PictureList "cambien"
      ProcessValue <- "Sensor_2"
   GraphicIOField "Graphic I/O field_19" at 569,214 size 25x48; PictureList "cambien"
      ProcessValue <- "Sensor_3"
   GraphicIOField "Graphic I/O field_20" at 667,214 size 25x48; PictureList "cambien"
      ProcessValue <- "Sensor_4"
   GraphicIOField "Graphic I/O field_21" at 761,214 size 25x48; PictureList "cambien"
      ProcessValue <- "Sensor_5"
   GraphicView "Graphic view_4" at 361,203 size 22x60; Picture "Graphic_14"
      Visibility <- "cylinder_1"
   GraphicView "Graphic view_2" at 449,203 size 22x94; Picture "Graphic_13"
      Visibility <- "cylinder_2"
   GraphicView "Graphic view_3" at 450,203 size 22x60; Picture "Graphic_14"
      Visibility <- "cylinder_2"
   GraphicView "Graphic view_5" at 548,203 size 22x94; Picture "Graphic_13"
      Visibility <- "cylinder_3"
   GraphicView "Graphic view_6" at 549,203 size 22x60; Picture "Graphic_14"
      Visibility <- "cylinder_3"
   GraphicView "Graphic view_7" at 641,203 size 22x94; Picture "Graphic_13"
      Visibility <- "cylinder_4"
   GraphicView "Graphic view_8" at 642,203 size 22x60; Picture "Graphic_14"
      Visibility <- "cylinder_4"
   GraphicView "Graphic view_9" at 738,203 size 22x94; Picture "Graphic_13"
      Visibility <- "cylinder_5"
   GraphicView "Graphic view_10" at 739,203 size 22x60; Picture "Graphic_14"
      Visibility <- "cylinder_5"
   TextField "Text field_9" at 360,176 size 69x23; Text 'Group 1'
   TextField "Text field_10" at 451,176 size 69x23; Text 'Group 2'
   TextField "Text field_11" at 543,176 size 69x23; Text 'Group 3'
   TextField "Text field_12" at 635,176 size 69x23; Text 'Group 4'
   TextField "Text field_13" at 727,176 size 69x23; Text 'Group 5'
   Circle "Circle_1" at 681,124 size 48x48
      Appearance <- "led_error"
   TextField "Text field_8" at 627,97 size 165x23; Text 'Error indicator light'
   Circle "Circle_2" at 503,124 size 48x48
      Appearance <- "state_to_webserver_state_emergency_stop"
   TextField "Text field_14" at 429,97 size 190x23; Text 'Lock run by Webserver'
   Circle "Circle_3" at 287,124 size 48x48
      Appearance <- "Data_webcam_state_camera"
   TextField "Text field_15" at 231,97 size 177x23; Text 'Connect with camera'
   GraphicIOField "Graphic I/O field_2" at 218,318 size 307x38; PictureList "bang_tai"
      ProcessValue <- "converyor"
   GraphicIOField "Graphic I/O field_5" at 476,317 size 323x38; PictureList "bang_tai"
      ProcessValue <- "converyor"

screen "Test_IO" 800x480, template "Template_1"
   TextField "Text field_1" at 338,141 size 124x22; Text 'TEST STATE I/O'
   TextField "Text field_2" at 350,113 size 100x23; Text 'MODE TEST'
   Rectangle "Rectangle_2" at 209,195 size 80x30
      Appearance <- "Sensor_1"
   Rectangle "Rectangle_3" at 209,241 size 80x30
      Appearance <- "Sensor_2"
   TextField "Text field_4" at 124,243 size 74x23; Text 'sensor2:'
   Rectangle "Rectangle_4" at 209,288 size 80x30
      Appearance <- "Sensor_3"
   TextField "Text field_5" at 124,291 size 74x23; Text 'sensor3:'
   Rectangle "Rectangle_5" at 209,335 size 80x30
      Appearance <- "Sensor_4"
   TextField "Text field_6" at 124,339 size 74x23; Text 'sensor4:'
   Rectangle "Rectangle_6" at 209,382 size 80x30
      Appearance <- "Sensor_5"
   TextField "Text field_7" at 124,387 size 74x23; Text 'sensor5:'
   Rectangle "Rectangle_7" at 209,429 size 80x30
      Appearance <- "Sensor_Detech"
   TextField "Text field_8" at 124,436 size 74x23; Text 'sensor6:'
   Rectangle "Rectangle_8" at 617,195 size 80x30
      Appearance <- "converyor"
   TextField "Text field_9" at 516,195 size 94x23; Text 'Converyor:'
   Rectangle "Rectangle_9" at 617,241 size 80x30
      Appearance <- "cylinder_1"
   TextField "Text field_10" at 516,243 size 93x23; Text 'Cylinder 1:'
   Rectangle "Rectangle_10" at 617,288 size 80x30
      Appearance <- "cylinder_2"
   Rectangle "Rectangle_11" at 617,335 size 80x30
      Appearance <- "cylinder_3"
   TextField "Text field_12" at 516,339 size 93x23; Text 'Cylinder 3:'
   Rectangle "Rectangle_12" at 617,382 size 80x30
      Appearance <- "cylinder_4"
   TextField "Text field_13" at 516,387 size 93x23; Text 'Cylinder 4:'
   Rectangle "Rectangle_13" at 617,429 size 80x30
      Appearance <- "cylinder_5"
   TextField "Text field_14" at 516,436 size 93x23; Text 'Cylinder 5:'
   TextField "Text field_11" at 515,291 size 93x23; Text 'Cylinder 2:'
   TextField "Text field_16" at 275,245 size 16x23; Text 'Text'
   TextField "Text field_3" at 129,195 size 74x23; Text 'sensor1:'

scheduled task "Showloginuser"
   on Action: function_f41c6f6c("Username")
*)